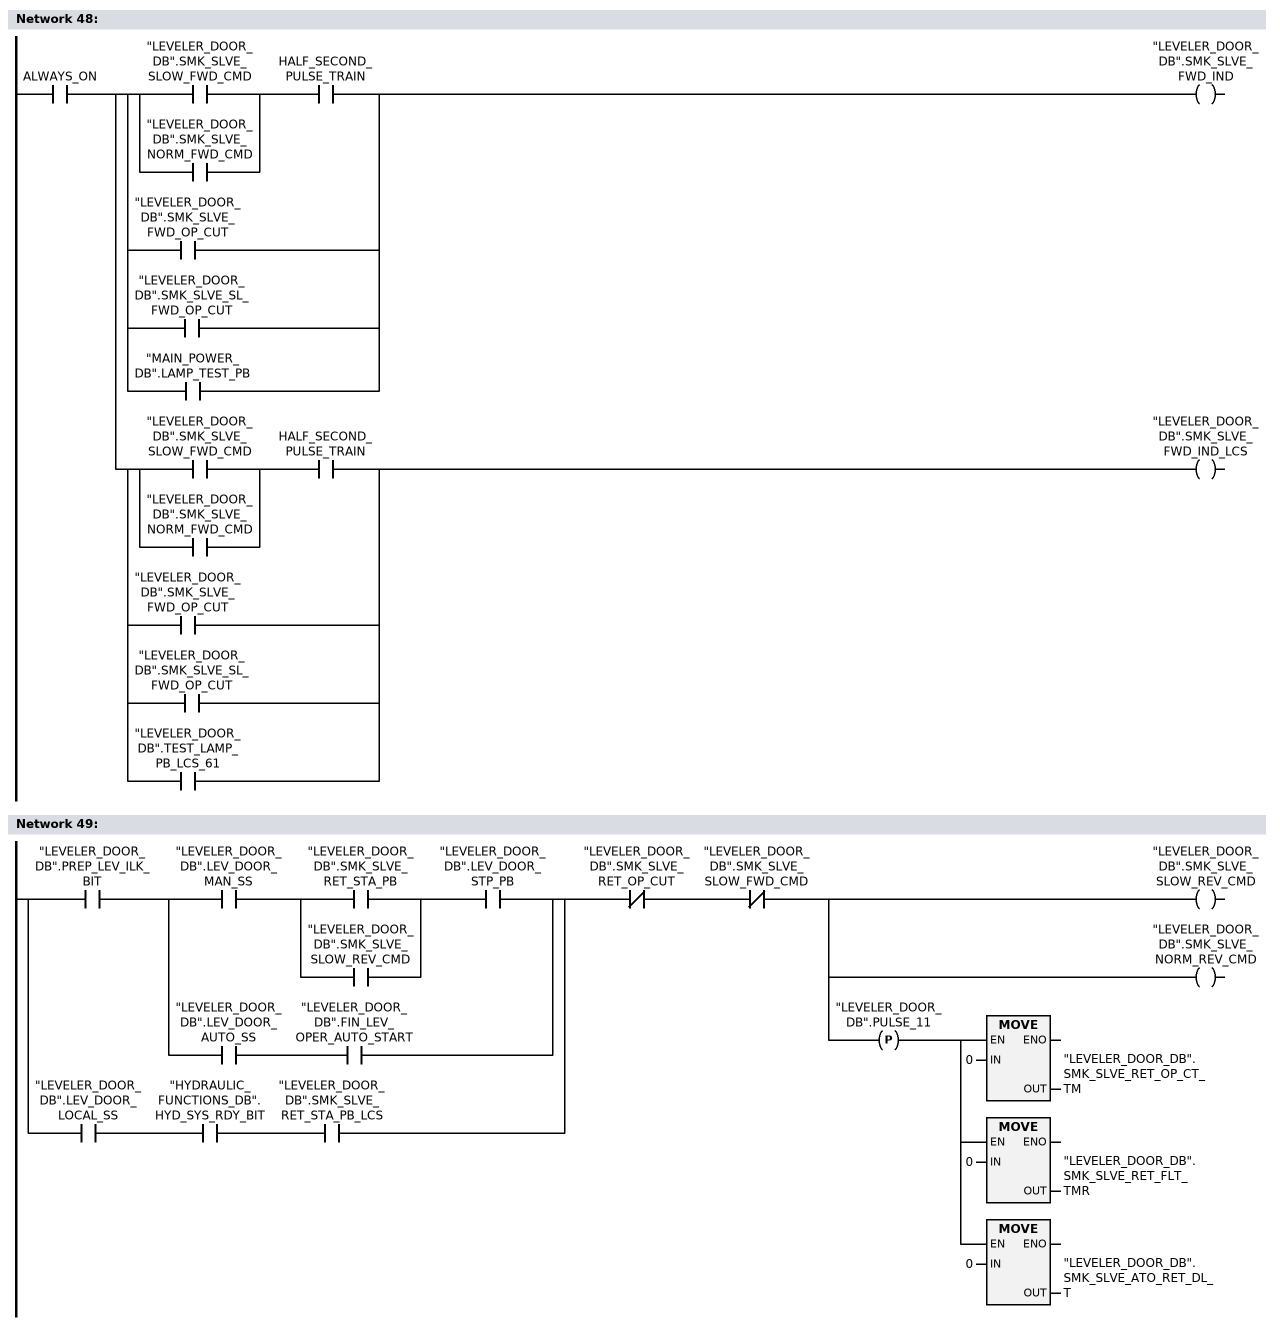
NETWORK
TITLE =
      A     "ALWAYS_ON";
      =     L 0.0;
      A     L 0.0;
      A(;
      A(;
      O     "LEVELER_DOOR_DB".SMK_SLVE_SLOW_FWD_CMD;
      O     "LEVELER_DOOR_DB".SMK_SLVE_NORM_FWD_CMD;
      );
      A     "HALF_SECOND_PULSE_TRAIN";
      O     "LEVELER_DOOR_DB".SMK_SLVE_FWD_OP_CUT;
      O     "LEVELER_DOOR_DB".SMK_SLVE_SL_FWD_OP_CUT;
      O     "MAIN_POWER_DB".LAMP_TEST_PB;
      );
      =     "LEVELER_DOOR_DB".SMK_SLVE_FWD_IND;
      A     L 0.0;
      A(;
      A(;
      O     "LEVELER_DOOR_DB".SMK_SLVE_SLOW_FWD_CMD;
      O     "LEVELER_DOOR_DB".SMK_SLVE_NORM_FWD_CMD;
      );
      A     "HALF_SECOND_PULSE_TRAIN";
      O     "LEVELER_DOOR_DB".SMK_SLVE_FWD_OP_CUT;
      O     "LEVELER_DOOR_DB".SMK_SLVE_SL_FWD_OP_CUT;
      O     "LEVELER_DOOR_DB".TEST_LAMP_PB_LCS_61;
      );
      =     "LEVELER_DOOR_DB".SMK_SLVE_FWD_IND_LCS;
NETWORK
TITLE =
      A(;
      A     "LEVELER_DOOR_DB".PREP_LEV_ILK_BIT;
      A(;
      A     "LEVELER_DOOR_DB".LEV_DOOR_MAN_SS;
      A(;
      O     "LEVELER_DOOR_DB".SMK_SLVE_RET_STA_PB;
      O     "LEVELER_DOOR_DB".SMK_SLVE_SLOW_REV_CMD;
      );
      A     "LEVELER_DOOR_DB".LEV_DOOR_STP_PB;
      O;
      A     "LEVELER_DOOR_DB".LEV_DOOR_AUTO_SS;
      A     "LEVELER_DOOR_DB".FIN_LEV_OPER_AUTO_START;
      );
      O;
      A     "LEVELER_DOOR_DB".LEV_DOOR_LOCAL_SS;
      A     "HYDRAULIC_FUNCTIONS_DB".HYD_SYS_RDY_BIT;
      A     "LEVELER_DOOR_DB".SMK_SLVE_RET_STA_PB_LCS;
      );
      AN    "LEVELER_DOOR_DB".SMK_SLVE_RET_OP_CUT;
      AN    "LEVELER_DOOR_DB".SMK_SLVE_SLOW_FWD_CMD;
      =     L 0.0;
      A     L 0.0;
      BLD   102;
      =     "LEVELER_DOOR_DB".SMK_SLVE_SLOW_REV_CMD;
      A     L 0.0;
      BLD   102;
      =     "LEVELER_DOOR_DB".SMK_SLVE_NORM_REV_CMD;
      A     L 0.0;
      FP    "LEVELER_DOOR_DB".PULSE_11;
      =     L 0.1;
      A     L 0.1;
      JNB   _030;
      L     0;
      T     "LEVELER_DOOR_DB".SMK_SLVE_RET_OP_CT_TM;
_030: NOP   0;
      A     L 0.1;
      JNB   _031;
      L     0;
      T     "LEVELER_DOOR_DB".SMK_SLVE_RET_FLT_TMR;
_031: NOP   0;
      A     L 0.1;
      JNB   _032;
      L     0;
      T     "LEVELER_DOOR_DB".SMK_SLVE_ATO_RET_DL_T;
_032: NOP   0;
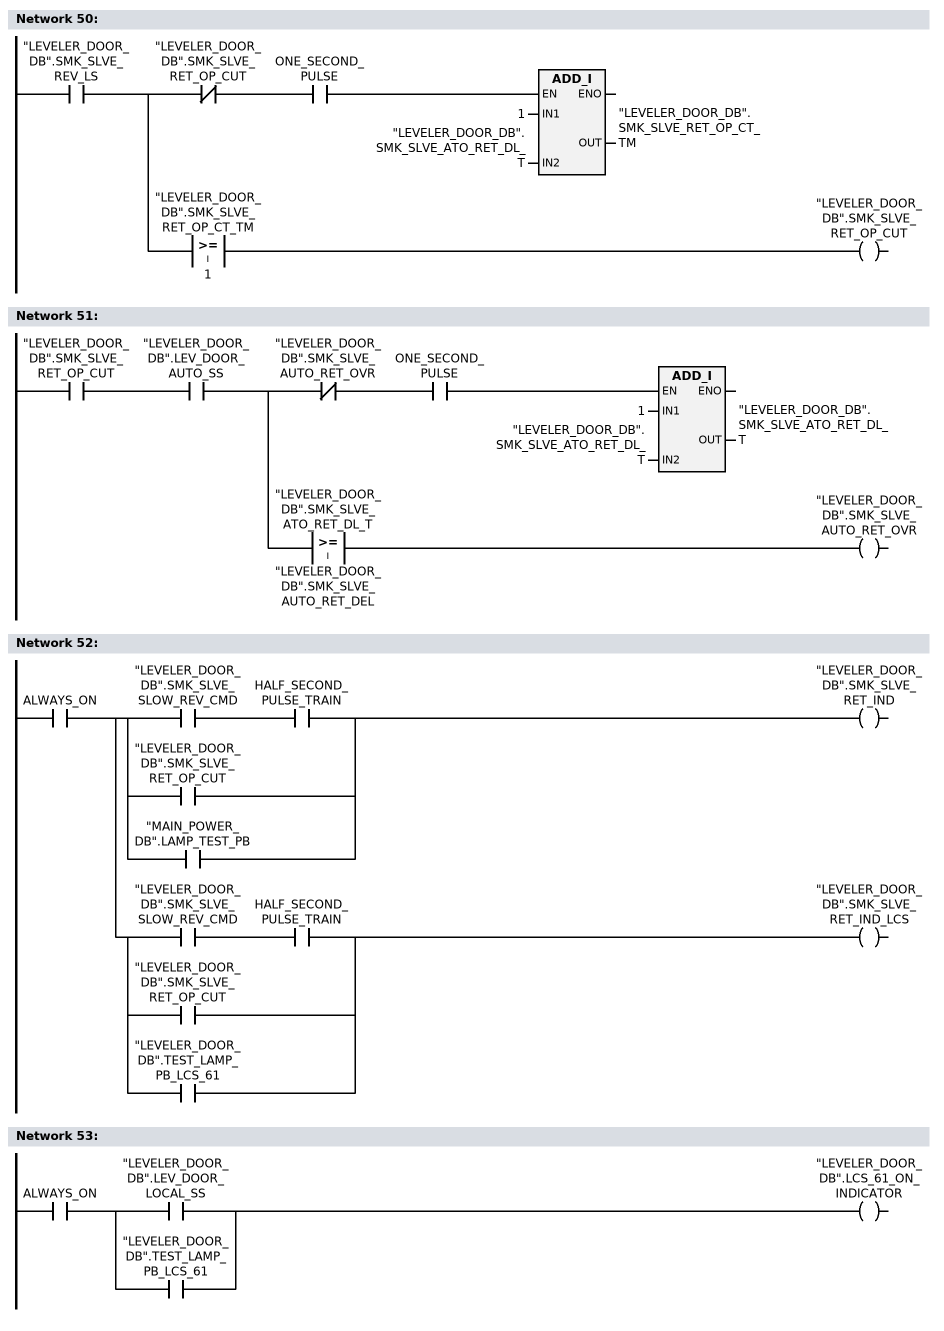
NETWORK
TITLE =
      A     "LEVELER_DOOR_DB".SMK_SLVE_REV_LS;
      =     L 0.0;
      A     L 0.0;
      AN    "LEVELER_DOOR_DB".SMK_SLVE_RET_OP_CUT;
      A     "ONE_SECOND_PULSE";
      JNB   _033;
      L     1;
      L     "LEVELER_DOOR_DB".SMK_SLVE_ATO_RET_DL_T;
      +I;
      T     "LEVELER_DOOR_DB".SMK_SLVE_RET_OP_CT_TM;
_033: NOP   0;
      A     L 0.0;
      A(;
      L     "LEVELER_DOOR_DB".SMK_SLVE_RET_OP_CT_TM;
      L     1;
      >=I;
      );
      =     "LEVELER_DOOR_DB".SMK_SLVE_RET_OP_CUT;
NETWORK
TITLE =
      A     "LEVELER_DOOR_DB".SMK_SLVE_RET_OP_CUT;
      A     "LEVELER_DOOR_DB".LEV_DOOR_AUTO_SS;
      =     L 0.0;
      A     L 0.0;
      AN    "LEVELER_DOOR_DB".SMK_SLVE_AUTO_RET_OVR;
      A     "ONE_SECOND_PULSE";
      JNB   _034;
      L     1;
      L     "LEVELER_DOOR_DB".SMK_SLVE_ATO_RET_DL_T;
      +I;
      T     "LEVELER_DOOR_DB".SMK_SLVE_ATO_RET_DL_T;
_034: NOP   0;
      A     L 0.0;
      A(;
      L     "LEVELER_DOOR_DB".SMK_SLVE_ATO_RET_DL_T;
      L     "LEVELER_DOOR_DB".SMK_SLVE_AUTO_RET_DEL;
      >=I;
      );
      =     "LEVELER_DOOR_DB".SMK_SLVE_AUTO_RET_OVR;
NETWORK
TITLE =
      A     "ALWAYS_ON";
      =     L 0.0;
      A     L 0.0;
      A(;
      A     "LEVELER_DOOR_DB".SMK_SLVE_SLOW_REV_CMD;
      A     "HALF_SECOND_PULSE_TRAIN";
      O     "LEVELER_DOOR_DB".SMK_SLVE_RET_OP_CUT;
      O     "MAIN_POWER_DB".LAMP_TEST_PB;
      );
      =     "LEVELER_DOOR_DB".SMK_SLVE_RET_IND;
      A     L 0.0;
      A(;
      A     "LEVELER_DOOR_DB".SMK_SLVE_SLOW_REV_CMD;
      A     "HALF_SECOND_PULSE_TRAIN";
      O     "LEVELER_DOOR_DB".SMK_SLVE_RET_OP_CUT;
      O     "LEVELER_DOOR_DB".TEST_LAMP_PB_LCS_61;
      );
      =     "LEVELER_DOOR_DB".SMK_SLVE_RET_IND_LCS;
NETWORK
TITLE =
      A     "ALWAYS_ON";
      A(;
      O     "LEVELER_DOOR_DB".LEV_DOOR_LOCAL_SS;
      O     "LEVELER_DOOR_DB".TEST_LAMP_PB_LCS_61;
      );
      =     "LEVELER_DOOR_DB".LCS_61_ON_INDICATOR;
END_FUNCTION

FUNCTION "TRAVEL_DRIVE" : VOID	// FC 7
AUTHOR : Kamillas
VERSION : 0.1
BEGIN
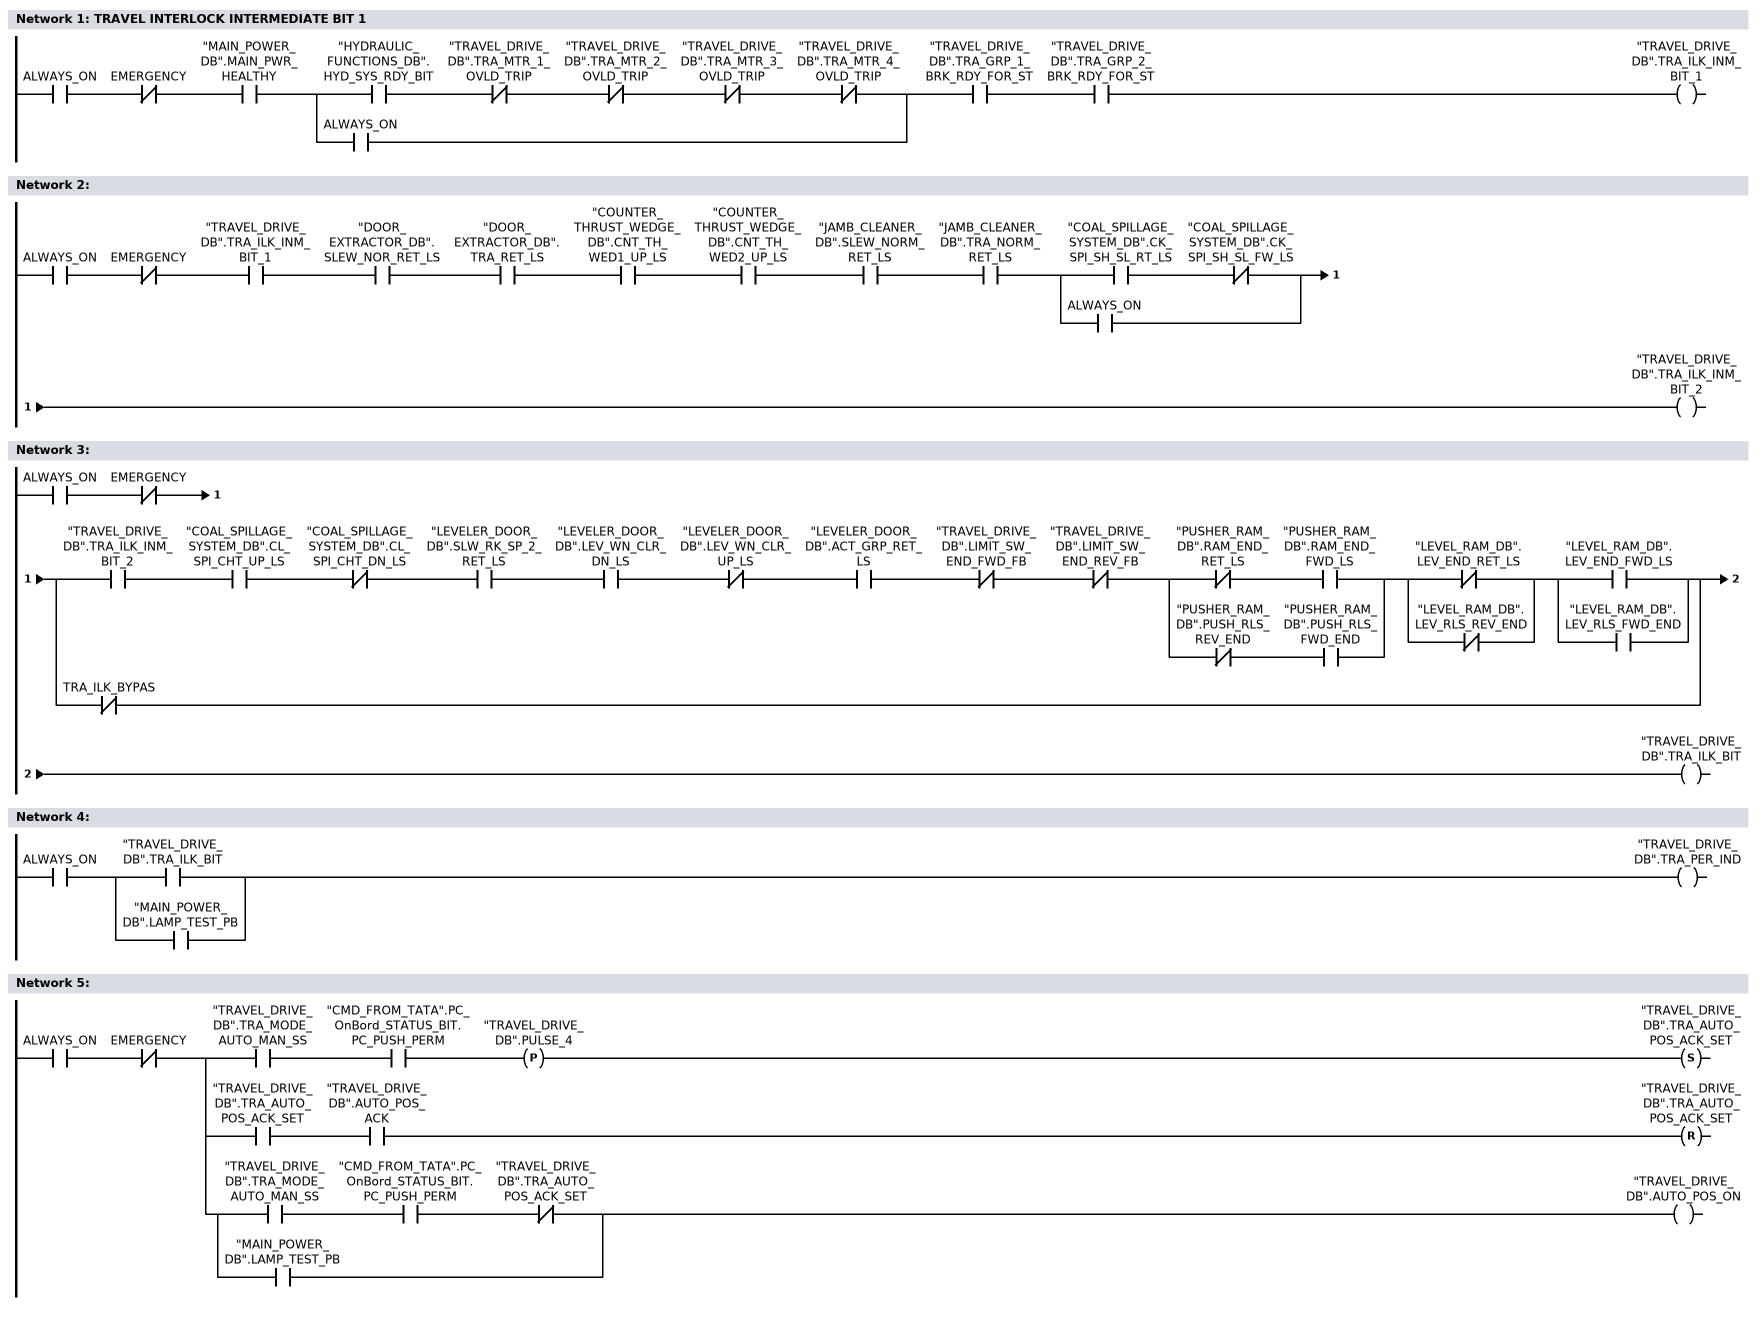
NETWORK
TITLE = TRAVEL INTERLOCK INTERMEDIATE BIT 1
      A     "ALWAYS_ON";
      AN    "EMERGENCY";
      A     "MAIN_POWER_DB".MAIN_PWR_HEALTHY;
      A(;
      A     "HYDRAULIC_FUNCTIONS_DB".HYD_SYS_RDY_BIT;
      AN    "TRAVEL_DRIVE_DB".TRA_MTR_1_OVLD_TRIP;
      AN    "TRAVEL_DRIVE_DB".TRA_MTR_2_OVLD_TRIP;
      AN    "TRAVEL_DRIVE_DB".TRA_MTR_3_OVLD_TRIP;
      AN    "TRAVEL_DRIVE_DB".TRA_MTR_4_OVLD_TRIP;
      O     "ALWAYS_ON";
      );
      A     "TRAVEL_DRIVE_DB".TRA_GRP_1_BRK_RDY_FOR_ST;
      A     "TRAVEL_DRIVE_DB".TRA_GRP_2_BRK_RDY_FOR_ST;
      =     "TRAVEL_DRIVE_DB".TRA_ILK_INM_BIT_1;
NETWORK
TITLE =
      A     "ALWAYS_ON";
      AN    "EMERGENCY";
      A     "TRAVEL_DRIVE_DB".TRA_ILK_INM_BIT_1;
      A     "DOOR_EXTRACTOR_DB".SLEW_NOR_RET_LS;
      A     "DOOR_EXTRACTOR_DB".TRA_RET_LS;
      A     "COUNTER_THRUST_WEDGE_DB".CNT_TH_WED1_UP_LS;
      A     "COUNTER_THRUST_WEDGE_DB".CNT_TH_WED2_UP_LS;
      A     "JAMB_CLEANER_DB".SLEW_NORM_RET_LS;
      A     "JAMB_CLEANER_DB".TRA_NORM_RET_LS;
      A(;
      A     "COAL_SPILLAGE_SYSTEM_DB".CK_SPI_SH_SL_RT_LS;
      AN    "COAL_SPILLAGE_SYSTEM_DB".CK_SPI_SH_SL_FW_LS;
      O     "ALWAYS_ON";
      );
      =     "TRAVEL_DRIVE_DB".TRA_ILK_INM_BIT_2;
NETWORK
TITLE =
      A     "ALWAYS_ON";
      AN    "EMERGENCY";
      A(;
      A     "TRAVEL_DRIVE_DB".TRA_ILK_INM_BIT_2;
      A     "COAL_SPILLAGE_SYSTEM_DB".CL_SPI_CHT_UP_LS;
      AN    "COAL_SPILLAGE_SYSTEM_DB".CL_SPI_CHT_DN_LS;
      A     "LEVELER_DOOR_DB".SLW_RK_SP_2_RET_LS;
      A     "LEVELER_DOOR_DB".LEV_WN_CLR_DN_LS;
      AN    "LEVELER_DOOR_DB".LEV_WN_CLR_UP_LS;
      A     "LEVELER_DOOR_DB".ACT_GRP_RET_LS;
      AN    "TRAVEL_DRIVE_DB".LIMIT_SW_END_FWD_FB;
      AN    "TRAVEL_DRIVE_DB".LIMIT_SW_END_REV_FB;
      A(;
      AN    "PUSHER_RAM_DB".RAM_END_RET_LS;
      A     "PUSHER_RAM_DB".RAM_END_FWD_LS;
      O;
      AN    "PUSHER_RAM_DB".PUSH_RLS_REV_END;
      A     "PUSHER_RAM_DB".PUSH_RLS_FWD_END;
      );
      A(;
      ON    "LEVEL_RAM_DB".LEV_END_RET_LS;
      ON    "LEVEL_RAM_DB".LEV_RLS_REV_END;
      );
      A(;
      O     "LEVEL_RAM_DB".LEV_END_FWD_LS;
      O     "LEVEL_RAM_DB".LEV_RLS_FWD_END;
      );
      ON    "TRA_ILK_BYPAS";
      );
      =     "TRAVEL_DRIVE_DB".TRA_ILK_BIT;
NETWORK
TITLE =
      A     "ALWAYS_ON";
      A(;
      O     "TRAVEL_DRIVE_DB".TRA_ILK_BIT;
      O     "MAIN_POWER_DB".LAMP_TEST_PB;
      );
      =     "TRAVEL_DRIVE_DB".TRA_PER_IND;
NETWORK
TITLE =
      A     "ALWAYS_ON";
      AN    "EMERGENCY";
      =     L 0.0;
      A     L 0.0;
      A     "TRAVEL_DRIVE_DB".TRA_MODE_AUTO_MAN_SS;
      A     "CMD_FROM_TATA".PC_OnBord_STATUS_BIT.PC_PUSH_PERM;
      FP    "TRAVEL_DRIVE_DB".PULSE_4;
      S     "TRAVEL_DRIVE_DB".TRA_AUTO_POS_ACK_SET;
      A     L 0.0;
      A     "TRAVEL_DRIVE_DB".TRA_AUTO_POS_ACK_SET;
      A     "TRAVEL_DRIVE_DB".AUTO_POS_ACK;
      R     "TRAVEL_DRIVE_DB".TRA_AUTO_POS_ACK_SET;
      A     L 0.0;
      A(;
      A     "TRAVEL_DRIVE_DB".TRA_MODE_AUTO_MAN_SS;
      A     "CMD_FROM_TATA".PC_OnBord_STATUS_BIT.PC_PUSH_PERM;
      AN    "TRAVEL_DRIVE_DB".TRA_AUTO_POS_ACK_SET;
      O     "MAIN_POWER_DB".LAMP_TEST_PB;
      );
      =     "TRAVEL_DRIVE_DB".AUTO_POS_ON;
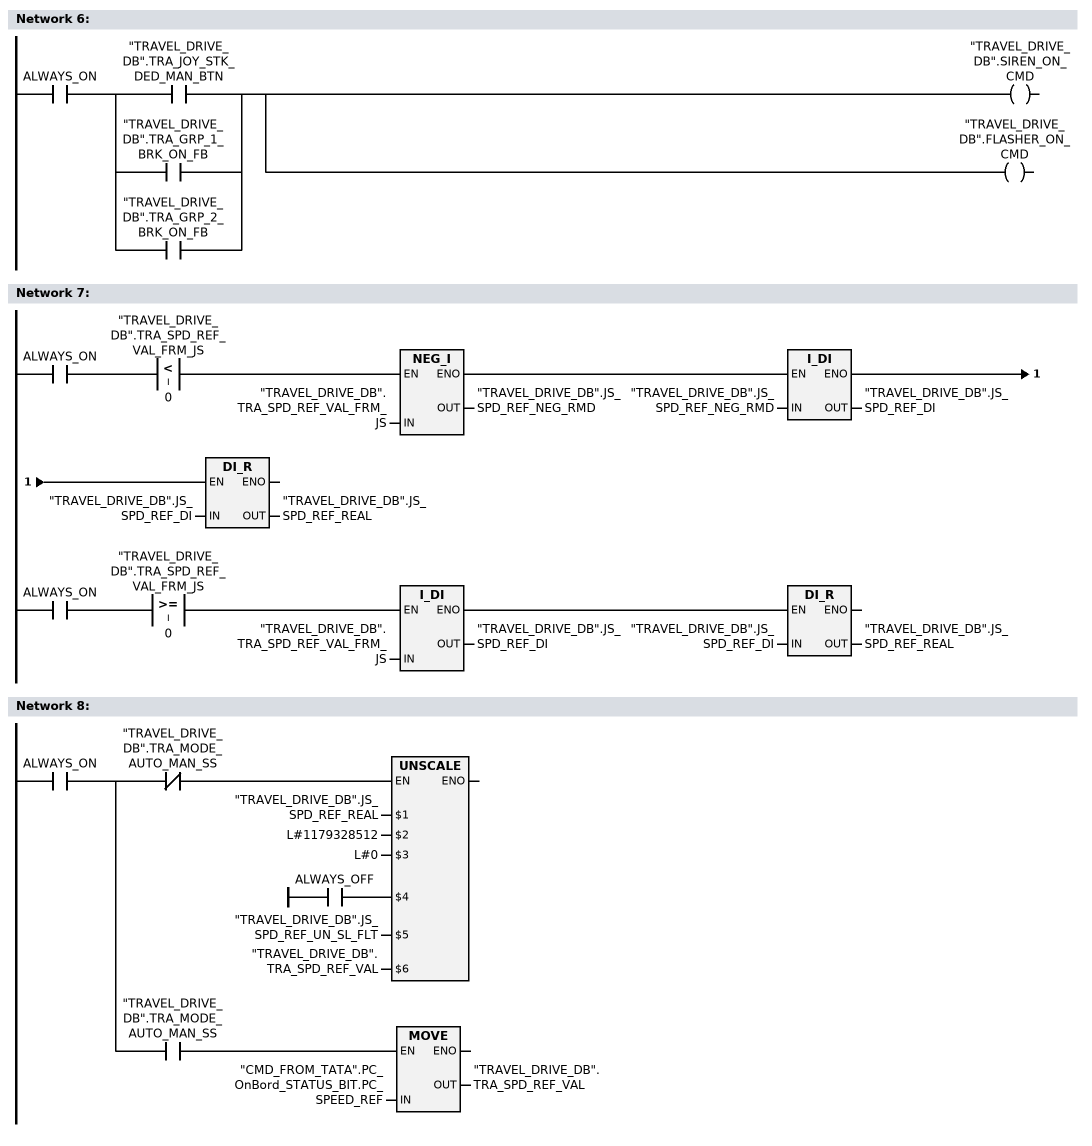
NETWORK
TITLE =
      A     "ALWAYS_ON";
      A(;
      O     "TRAVEL_DRIVE_DB".TRA_JOY_STK_DED_MAN_BTN;
      O     "TRAVEL_DRIVE_DB".TRA_GRP_1_BRK_ON_FB;
      O     "TRAVEL_DRIVE_DB".TRA_GRP_2_BRK_ON_FB;
      );
      =     "TRAVEL_DRIVE_DB".SIREN_ON_CMD;
      =     "TRAVEL_DRIVE_DB".FLASHER_ON_CMD;
NETWORK
TITLE =
      A     "ALWAYS_ON";
      =     L 0.0;
      A(;
      A(;
      A     L 0.0;
      A(;
      L     "TRAVEL_DRIVE_DB".TRA_SPD_REF_VAL_FRM_JS;
      L     0;
      <I;
      );
      JNB   _001;
      L     "TRAVEL_DRIVE_DB".TRA_SPD_REF_VAL_FRM_JS;
      NEGI;
      T     "TRAVEL_DRIVE_DB".JS_SPD_REF_NEG_RMD;
      AN    OV;
      SAVE;
      CLR;
_001: A     BR;
      );
      JNB   _002;
      L     "TRAVEL_DRIVE_DB".JS_SPD_REF_NEG_RMD;
      ITD;
      T     "TRAVEL_DRIVE_DB".JS_SPD_REF_DI;
      SET;
      SAVE;
      CLR;
_002: A     BR;
      );
      JNB   _003;
      L     "TRAVEL_DRIVE_DB".JS_SPD_REF_DI;
      DTR;
      T     "TRAVEL_DRIVE_DB".JS_SPD_REF_REAL;
_003: NOP   0;
      A(;
      A     L 0.0;
      A(;
      L     "TRAVEL_DRIVE_DB".TRA_SPD_REF_VAL_FRM_JS;
      L     0;
      >=I;
      );
      JNB   _004;
      L     "TRAVEL_DRIVE_DB".TRA_SPD_REF_VAL_FRM_JS;
      ITD;
      T     "TRAVEL_DRIVE_DB".JS_SPD_REF_DI;
      SET;
      SAVE;
      CLR;
_004: A     BR;
      );
      JNB   _005;
      L     "TRAVEL_DRIVE_DB".JS_SPD_REF_DI;
      DTR;
      T     "TRAVEL_DRIVE_DB".JS_SPD_REF_REAL;
_005: NOP   0;
NETWORK
TITLE =
      A     "ALWAYS_ON";
      =     L 0.0;
      A     "ALWAYS_OFF";
      =     L 0.1;
      BLD   103;
      A     L 0.0;
      AN    "TRAVEL_DRIVE_DB".TRA_MODE_AUTO_MAN_SS;
      JNB   _006;
      CALL  "UNSCALE" (
           $1                       := "TRAVEL_DRIVE_DB".JS_SPD_REF_REAL,
           $2                       := L#1179328512,
           $3                       := L#0,
           $4                       := L 0.1,
           $5                       := "TRAVEL_DRIVE_DB".JS_SPD_REF_UN_SL_FLT,
           $6                       := "TRAVEL_DRIVE_DB".TRA_SPD_REF_VAL);
_006: NOP   0;
      A     L 0.0;
      A     "TRAVEL_DRIVE_DB".TRA_MODE_AUTO_MAN_SS;
      JNB   _007;
      L     "CMD_FROM_TATA".PC_OnBord_STATUS_BIT.PC_SPEED_REF;
      T     "TRAVEL_DRIVE_DB".TRA_SPD_REF_VAL;
_007: NOP   0;
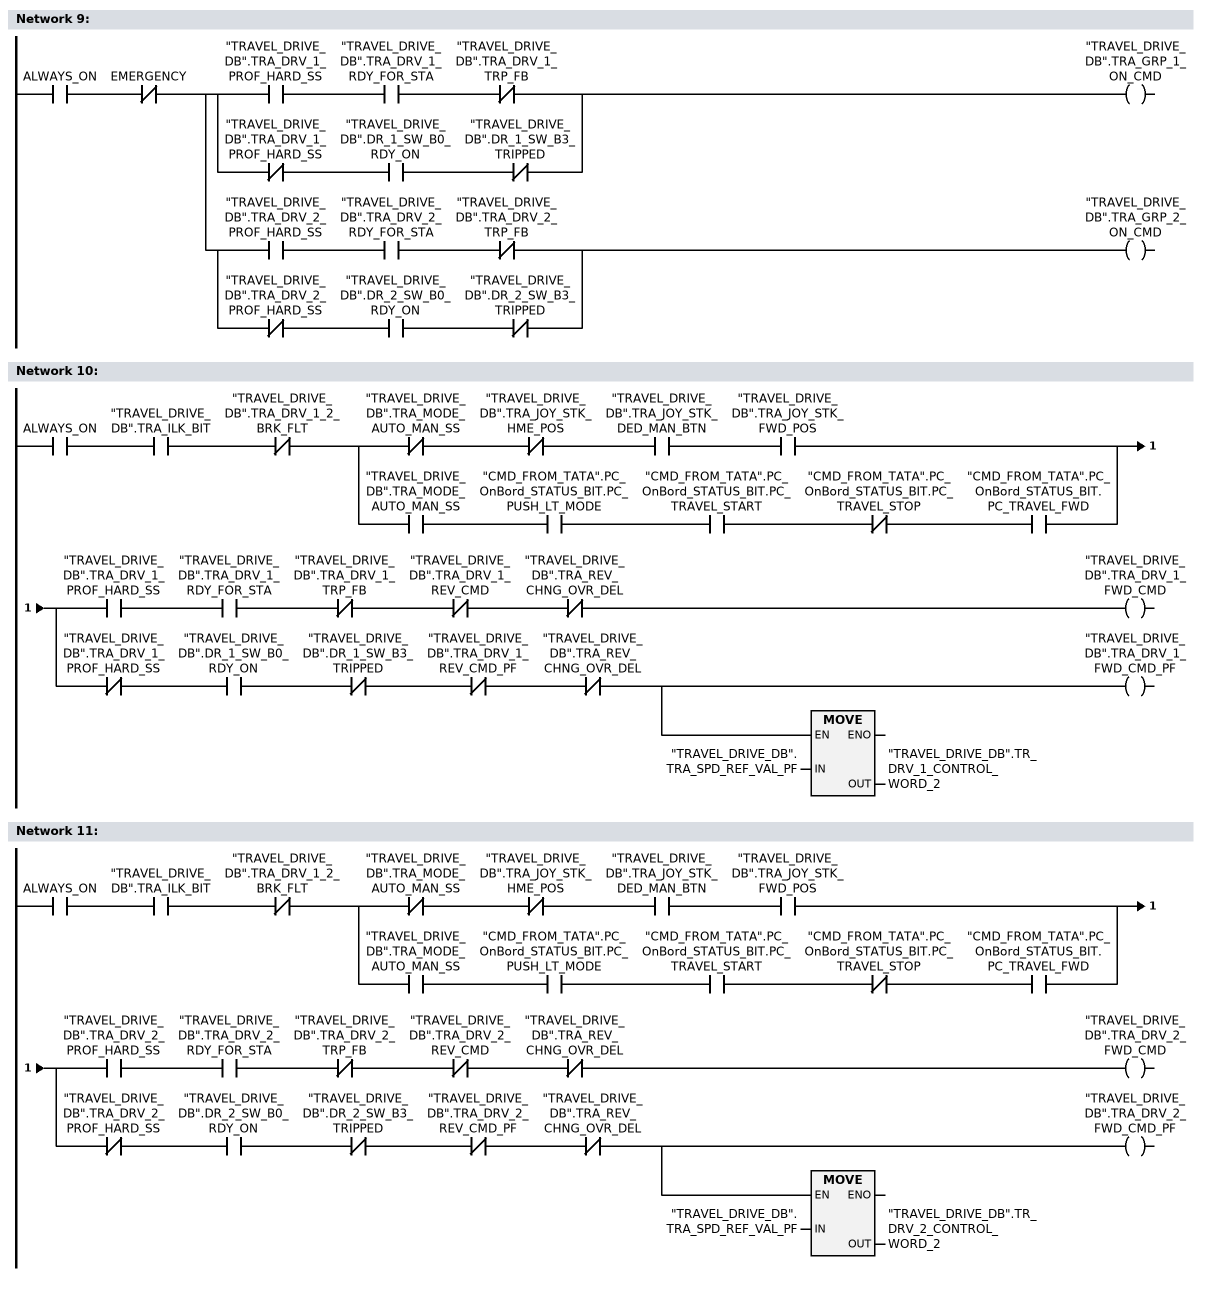
NETWORK
TITLE =
      A     "ALWAYS_ON";
      AN    "EMERGENCY";
      =     L 0.0;
      A     L 0.0;
      A(;
      A     "TRAVEL_DRIVE_DB".TRA_DRV_1_PROF_HARD_SS;
      A     "TRAVEL_DRIVE_DB".TRA_DRV_1_RDY_FOR_STA;
      AN    "TRAVEL_DRIVE_DB".TRA_DRV_1_TRP_FB;
      O;
      AN    "TRAVEL_DRIVE_DB".TRA_DRV_1_PROF_HARD_SS;
      A     "TRAVEL_DRIVE_DB".DR_1_SW_B0_RDY_ON;
      AN    "TRAVEL_DRIVE_DB".DR_1_SW_B3_TRIPPED;
      );
      =     "TRAVEL_DRIVE_DB".TRA_GRP_1_ON_CMD;
      A     L 0.0;
      A(;
      A     "TRAVEL_DRIVE_DB".TRA_DRV_2_PROF_HARD_SS;
      A     "TRAVEL_DRIVE_DB".TRA_DRV_2_RDY_FOR_STA;
      AN    "TRAVEL_DRIVE_DB".TRA_DRV_2_TRP_FB;
      O;
      AN    "TRAVEL_DRIVE_DB".TRA_DRV_2_PROF_HARD_SS;
      A     "TRAVEL_DRIVE_DB".DR_2_SW_B0_RDY_ON;
      AN    "TRAVEL_DRIVE_DB".DR_2_SW_B3_TRIPPED;
      );
      =     "TRAVEL_DRIVE_DB".TRA_GRP_2_ON_CMD;
NETWORK
TITLE =
      A     "ALWAYS_ON";
      A     "TRAVEL_DRIVE_DB".TRA_ILK_BIT;
      AN    "TRAVEL_DRIVE_DB".TRA_DRV_1_2_BRK_FLT;
      A(;
      AN    "TRAVEL_DRIVE_DB".TRA_MODE_AUTO_MAN_SS;
      AN    "TRAVEL_DRIVE_DB".TRA_JOY_STK_HME_POS;
      A     "TRAVEL_DRIVE_DB".TRA_JOY_STK_DED_MAN_BTN;
      A     "TRAVEL_DRIVE_DB".TRA_JOY_STK_FWD_POS;
      O;
      A     "TRAVEL_DRIVE_DB".TRA_MODE_AUTO_MAN_SS;
      A     "CMD_FROM_TATA".PC_OnBord_STATUS_BIT.PC_PUSH_LT_MODE;
      A     "CMD_FROM_TATA".PC_OnBord_STATUS_BIT.PC_TRAVEL_START;
      AN    "CMD_FROM_TATA".PC_OnBord_STATUS_BIT.PC_TRAVEL_STOP;
      A     "CMD_FROM_TATA".PC_OnBord_STATUS_BIT.PC_TRAVEL_FWD;
      );
      =     L 0.0;
      A     L 0.0;
      A     "TRAVEL_DRIVE_DB".TRA_DRV_1_PROF_HARD_SS;
      A     "TRAVEL_DRIVE_DB".TRA_DRV_1_RDY_FOR_STA;
      AN    "TRAVEL_DRIVE_DB".TRA_DRV_1_TRP_FB;
      AN    "TRAVEL_DRIVE_DB".TRA_DRV_1_REV_CMD;
      AN    "TRAVEL_DRIVE_DB".TRA_REV_CHNG_OVR_DEL;
      =     "TRAVEL_DRIVE_DB".TRA_DRV_1_FWD_CMD;
      A     L 0.0;
      AN    "TRAVEL_DRIVE_DB".TRA_DRV_1_PROF_HARD_SS;
      A     "TRAVEL_DRIVE_DB".DR_1_SW_B0_RDY_ON;
      AN    "TRAVEL_DRIVE_DB".DR_1_SW_B3_TRIPPED;
      AN    "TRAVEL_DRIVE_DB".TRA_DRV_1_REV_CMD_PF;
      AN    "TRAVEL_DRIVE_DB".TRA_REV_CHNG_OVR_DEL;
      =     L 0.1;
      A     L 0.1;
      BLD   102;
      =     "TRAVEL_DRIVE_DB".TRA_DRV_1_FWD_CMD_PF;
      A     L 0.1;
      JNB   _008;
      L     "TRAVEL_DRIVE_DB".TRA_SPD_REF_VAL_PF;
      T     "TRAVEL_DRIVE_DB".TR_DRV_1_CONTROL_WORD_2;
_008: NOP   0;
NETWORK
TITLE =
      A     "ALWAYS_ON";
      A     "TRAVEL_DRIVE_DB".TRA_ILK_BIT;
      AN    "TRAVEL_DRIVE_DB".TRA_DRV_1_2_BRK_FLT;
      A(;
      AN    "TRAVEL_DRIVE_DB".TRA_MODE_AUTO_MAN_SS;
      AN    "TRAVEL_DRIVE_DB".TRA_JOY_STK_HME_POS;
      A     "TRAVEL_DRIVE_DB".TRA_JOY_STK_DED_MAN_BTN;
      A     "TRAVEL_DRIVE_DB".TRA_JOY_STK_FWD_POS;
      O;
      A     "TRAVEL_DRIVE_DB".TRA_MODE_AUTO_MAN_SS;
      A     "CMD_FROM_TATA".PC_OnBord_STATUS_BIT.PC_PUSH_LT_MODE;
      A     "CMD_FROM_TATA".PC_OnBord_STATUS_BIT.PC_TRAVEL_START;
      AN    "CMD_FROM_TATA".PC_OnBord_STATUS_BIT.PC_TRAVEL_STOP;
      A     "CMD_FROM_TATA".PC_OnBord_STATUS_BIT.PC_TRAVEL_FWD;
      );
      =     L 0.0;
      A     L 0.0;
      A     "TRAVEL_DRIVE_DB".TRA_DRV_2_PROF_HARD_SS;
      A     "TRAVEL_DRIVE_DB".TRA_DRV_2_RDY_FOR_STA;
      AN    "TRAVEL_DRIVE_DB".TRA_DRV_2_TRP_FB;
      AN    "TRAVEL_DRIVE_DB".TRA_DRV_2_REV_CMD;
      AN    "TRAVEL_DRIVE_DB".TRA_REV_CHNG_OVR_DEL;
      =     "TRAVEL_DRIVE_DB".TRA_DRV_2_FWD_CMD;
      A     L 0.0;
      AN    "TRAVEL_DRIVE_DB".TRA_DRV_2_PROF_HARD_SS;
      A     "TRAVEL_DRIVE_DB".DR_2_SW_B0_RDY_ON;
      AN    "TRAVEL_DRIVE_DB".DR_2_SW_B3_TRIPPED;
      AN    "TRAVEL_DRIVE_DB".TRA_DRV_2_REV_CMD_PF;
      AN    "TRAVEL_DRIVE_DB".TRA_REV_CHNG_OVR_DEL;
      =     L 0.1;
      A     L 0.1;
      BLD   102;
      =     "TRAVEL_DRIVE_DB".TRA_DRV_2_FWD_CMD_PF;
      A     L 0.1;
      JNB   _009;
      L     "TRAVEL_DRIVE_DB".TRA_SPD_REF_VAL_PF;
      T     "TRAVEL_DRIVE_DB".TR_DRV_2_CONTROL_WORD_2;
_009: NOP   0;
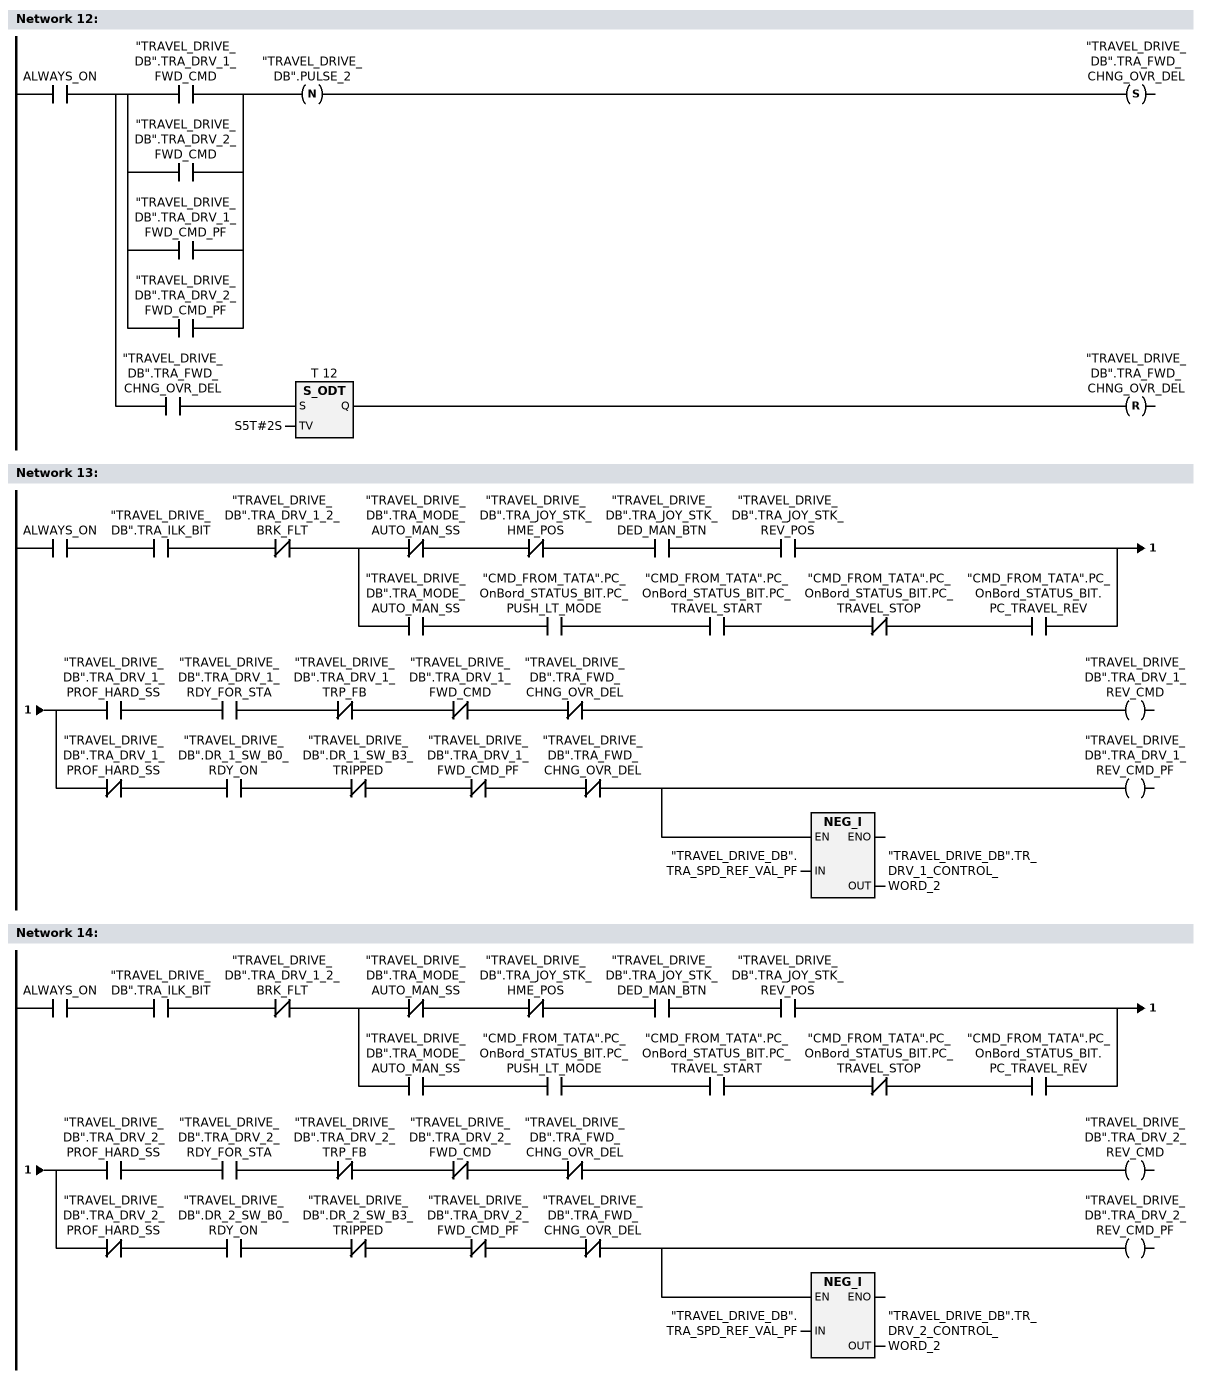
NETWORK
TITLE =
      A     "ALWAYS_ON";
      =     L 0.0;
      A     L 0.0;
      A(;
      O     "TRAVEL_DRIVE_DB".TRA_DRV_1_FWD_CMD;
      O     "TRAVEL_DRIVE_DB".TRA_DRV_2_FWD_CMD;
      O     "TRAVEL_DRIVE_DB".TRA_DRV_1_FWD_CMD_PF;
      O     "TRAVEL_DRIVE_DB".TRA_DRV_2_FWD_CMD_PF;
      );
      FN    "TRAVEL_DRIVE_DB".PULSE_2;
      S     "TRAVEL_DRIVE_DB".TRA_FWD_CHNG_OVR_DEL;
      A     L 0.0;
      A     "TRAVEL_DRIVE_DB".TRA_FWD_CHNG_OVR_DEL;
      L     S5T#2S;
      SD    T 12;
      NOP   0;
      NOP   0;
      NOP   0;
      A     T 12;
      R     "TRAVEL_DRIVE_DB".TRA_FWD_CHNG_OVR_DEL;
NETWORK
TITLE =
      A     "ALWAYS_ON";
      A     "TRAVEL_DRIVE_DB".TRA_ILK_BIT;
      AN    "TRAVEL_DRIVE_DB".TRA_DRV_1_2_BRK_FLT;
      A(;
      AN    "TRAVEL_DRIVE_DB".TRA_MODE_AUTO_MAN_SS;
      AN    "TRAVEL_DRIVE_DB".TRA_JOY_STK_HME_POS;
      A     "TRAVEL_DRIVE_DB".TRA_JOY_STK_DED_MAN_BTN;
      A     "TRAVEL_DRIVE_DB".TRA_JOY_STK_REV_POS;
      O;
      A     "TRAVEL_DRIVE_DB".TRA_MODE_AUTO_MAN_SS;
      A     "CMD_FROM_TATA".PC_OnBord_STATUS_BIT.PC_PUSH_LT_MODE;
      A     "CMD_FROM_TATA".PC_OnBord_STATUS_BIT.PC_TRAVEL_START;
      AN    "CMD_FROM_TATA".PC_OnBord_STATUS_BIT.PC_TRAVEL_STOP;
      A     "CMD_FROM_TATA".PC_OnBord_STATUS_BIT.PC_TRAVEL_REV;
      );
      =     L 0.0;
      A     L 0.0;
      A     "TRAVEL_DRIVE_DB".TRA_DRV_1_PROF_HARD_SS;
      A     "TRAVEL_DRIVE_DB".TRA_DRV_1_RDY_FOR_STA;
      AN    "TRAVEL_DRIVE_DB".TRA_DRV_1_TRP_FB;
      AN    "TRAVEL_DRIVE_DB".TRA_DRV_1_FWD_CMD;
      AN    "TRAVEL_DRIVE_DB".TRA_FWD_CHNG_OVR_DEL;
      =     "TRAVEL_DRIVE_DB".TRA_DRV_1_REV_CMD;
      A     L 0.0;
      AN    "TRAVEL_DRIVE_DB".TRA_DRV_1_PROF_HARD_SS;
      A     "TRAVEL_DRIVE_DB".DR_1_SW_B0_RDY_ON;
      AN    "TRAVEL_DRIVE_DB".DR_1_SW_B3_TRIPPED;
      AN    "TRAVEL_DRIVE_DB".TRA_DRV_1_FWD_CMD_PF;
      AN    "TRAVEL_DRIVE_DB".TRA_FWD_CHNG_OVR_DEL;
      =     L 0.1;
      A     L 0.1;
      BLD   102;
      =     "TRAVEL_DRIVE_DB".TRA_DRV_1_REV_CMD_PF;
      A     L 0.1;
      JNB   _00a;
      L     "TRAVEL_DRIVE_DB".TRA_SPD_REF_VAL_PF;
      NEGI;
      T     "TRAVEL_DRIVE_DB".TR_DRV_1_CONTROL_WORD_2;
_00a: NOP   0;
NETWORK
TITLE =
      A     "ALWAYS_ON";
      A     "TRAVEL_DRIVE_DB".TRA_ILK_BIT;
      AN    "TRAVEL_DRIVE_DB".TRA_DRV_1_2_BRK_FLT;
      A(;
      AN    "TRAVEL_DRIVE_DB".TRA_MODE_AUTO_MAN_SS;
      AN    "TRAVEL_DRIVE_DB".TRA_JOY_STK_HME_POS;
      A     "TRAVEL_DRIVE_DB".TRA_JOY_STK_DED_MAN_BTN;
      A     "TRAVEL_DRIVE_DB".TRA_JOY_STK_REV_POS;
      O;
      A     "TRAVEL_DRIVE_DB".TRA_MODE_AUTO_MAN_SS;
      A     "CMD_FROM_TATA".PC_OnBord_STATUS_BIT.PC_PUSH_LT_MODE;
      A     "CMD_FROM_TATA".PC_OnBord_STATUS_BIT.PC_TRAVEL_START;
      AN    "CMD_FROM_TATA".PC_OnBord_STATUS_BIT.PC_TRAVEL_STOP;
      A     "CMD_FROM_TATA".PC_OnBord_STATUS_BIT.PC_TRAVEL_REV;
      );
      =     L 0.0;
      A     L 0.0;
      A     "TRAVEL_DRIVE_DB".TRA_DRV_2_PROF_HARD_SS;
      A     "TRAVEL_DRIVE_DB".TRA_DRV_2_RDY_FOR_STA;
      AN    "TRAVEL_DRIVE_DB".TRA_DRV_2_TRP_FB;
      AN    "TRAVEL_DRIVE_DB".TRA_DRV_2_FWD_CMD;
      AN    "TRAVEL_DRIVE_DB".TRA_FWD_CHNG_OVR_DEL;
      =     "TRAVEL_DRIVE_DB".TRA_DRV_2_REV_CMD;
      A     L 0.0;
      AN    "TRAVEL_DRIVE_DB".TRA_DRV_2_PROF_HARD_SS;
      A     "TRAVEL_DRIVE_DB".DR_2_SW_B0_RDY_ON;
      AN    "TRAVEL_DRIVE_DB".DR_2_SW_B3_TRIPPED;
      AN    "TRAVEL_DRIVE_DB".TRA_DRV_2_FWD_CMD_PF;
      AN    "TRAVEL_DRIVE_DB".TRA_FWD_CHNG_OVR_DEL;
      =     L 0.1;
      A     L 0.1;
      BLD   102;
      =     "TRAVEL_DRIVE_DB".TRA_DRV_2_REV_CMD_PF;
      A     L 0.1;
      JNB   _00b;
      L     "TRAVEL_DRIVE_DB".TRA_SPD_REF_VAL_PF;
      NEGI;
      T     "TRAVEL_DRIVE_DB".TR_DRV_2_CONTROL_WORD_2;
_00b: NOP   0;
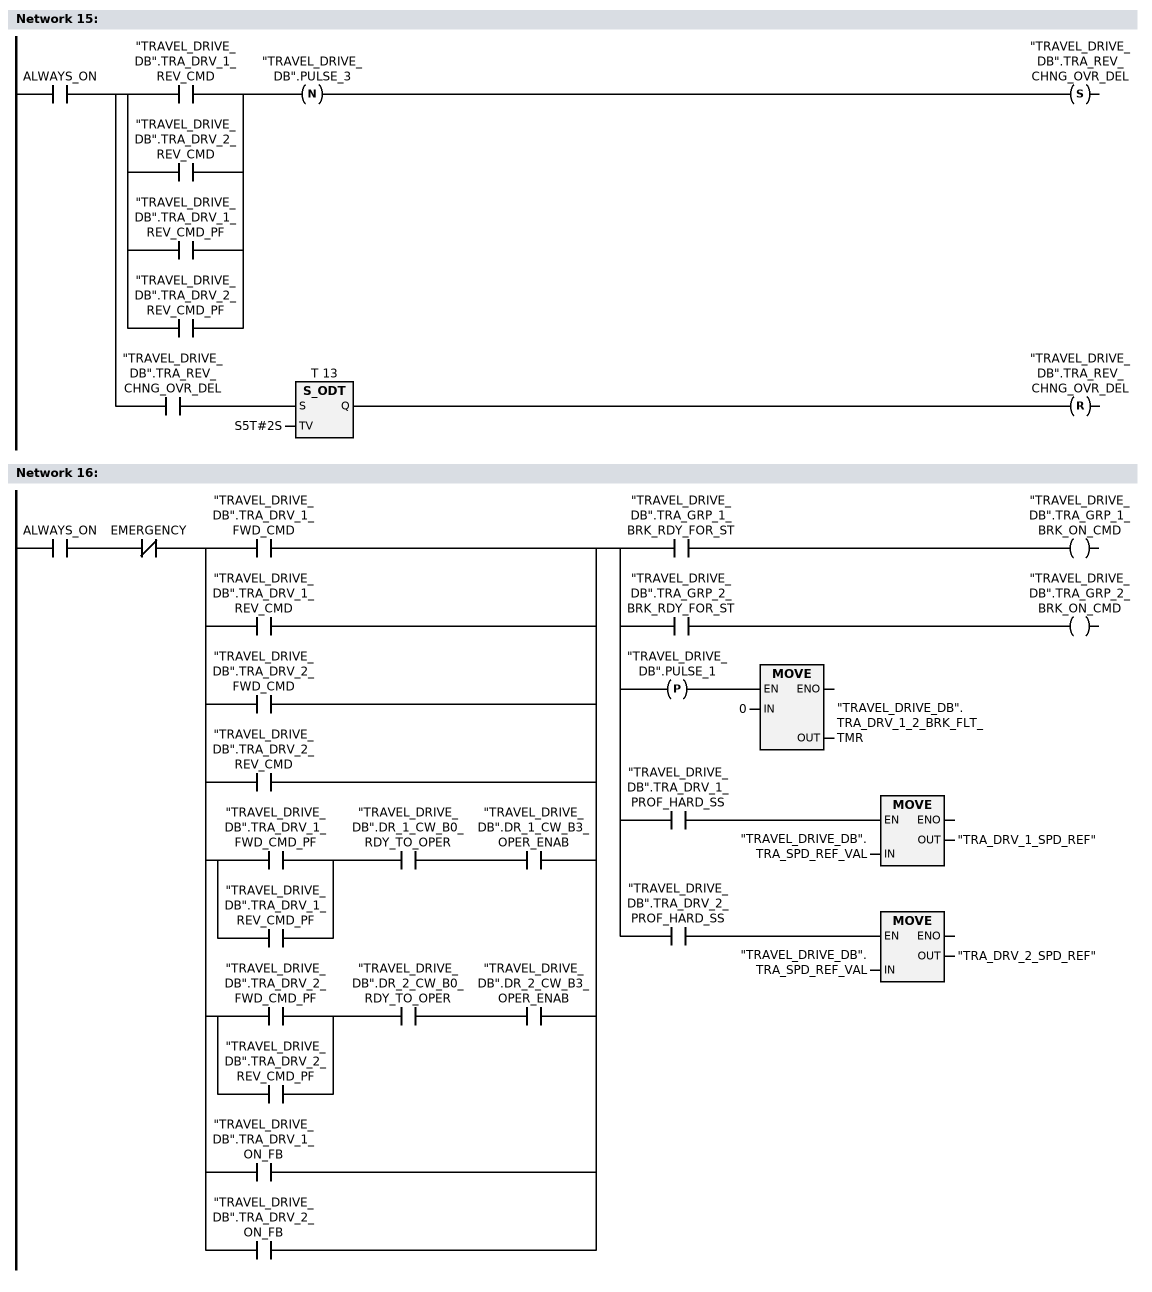
NETWORK
TITLE =
      A     "ALWAYS_ON";
      =     L 0.0;
      A     L 0.0;
      A(;
      O     "TRAVEL_DRIVE_DB".TRA_DRV_1_REV_CMD;
      O     "TRAVEL_DRIVE_DB".TRA_DRV_2_REV_CMD;
      O     "TRAVEL_DRIVE_DB".TRA_DRV_1_REV_CMD_PF;
      O     "TRAVEL_DRIVE_DB".TRA_DRV_2_REV_CMD_PF;
      );
      FN    "TRAVEL_DRIVE_DB".PULSE_3;
      S     "TRAVEL_DRIVE_DB".TRA_REV_CHNG_OVR_DEL;
      A     L 0.0;
      A     "TRAVEL_DRIVE_DB".TRA_REV_CHNG_OVR_DEL;
      L     S5T#2S;
      SD    T 13;
      NOP   0;
      NOP   0;
      NOP   0;
      A     T 13;
      R     "TRAVEL_DRIVE_DB".TRA_REV_CHNG_OVR_DEL;
NETWORK
TITLE =
      A     "ALWAYS_ON";
      AN    "EMERGENCY";
      A(;
      O     "TRAVEL_DRIVE_DB".TRA_DRV_1_FWD_CMD;
      O     "TRAVEL_DRIVE_DB".TRA_DRV_1_REV_CMD;
      O     "TRAVEL_DRIVE_DB".TRA_DRV_2_FWD_CMD;
      O     "TRAVEL_DRIVE_DB".TRA_DRV_2_REV_CMD;
      O;
      A(;
      O     "TRAVEL_DRIVE_DB".TRA_DRV_1_FWD_CMD_PF;
      O     "TRAVEL_DRIVE_DB".TRA_DRV_1_REV_CMD_PF;
      );
      A     "TRAVEL_DRIVE_DB".DR_1_CW_B0_RDY_TO_OPER;
      A     "TRAVEL_DRIVE_DB".DR_1_CW_B3_OPER_ENAB;
      O;
      A(;
      O     "TRAVEL_DRIVE_DB".TRA_DRV_2_FWD_CMD_PF;
      O     "TRAVEL_DRIVE_DB".TRA_DRV_2_REV_CMD_PF;
      );
      A     "TRAVEL_DRIVE_DB".DR_2_CW_B0_RDY_TO_OPER;
      A     "TRAVEL_DRIVE_DB".DR_2_CW_B3_OPER_ENAB;
      O     "TRAVEL_DRIVE_DB".TRA_DRV_1_ON_FB;
      O     "TRAVEL_DRIVE_DB".TRA_DRV_2_ON_FB;
      );
      =     L 0.0;
      A     L 0.0;
      A     "TRAVEL_DRIVE_DB".TRA_GRP_1_BRK_RDY_FOR_ST;
      =     "TRAVEL_DRIVE_DB".TRA_GRP_1_BRK_ON_CMD;
      A     L 0.0;
      A     "TRAVEL_DRIVE_DB".TRA_GRP_2_BRK_RDY_FOR_ST;
      =     "TRAVEL_DRIVE_DB".TRA_GRP_2_BRK_ON_CMD;
      A     L 0.0;
      FP    "TRAVEL_DRIVE_DB".PULSE_1;
      JNB   _00c;
      L     0;
      T     "TRAVEL_DRIVE_DB".TRA_DRV_1_2_BRK_FLT_TMR;
_00c: NOP   0;
      A     L 0.0;
      A     "TRAVEL_DRIVE_DB".TRA_DRV_1_PROF_HARD_SS;
      JNB   _00d;
      L     "TRAVEL_DRIVE_DB".TRA_SPD_REF_VAL;
      T     "TRA_DRV_1_SPD_REF";
_00d: NOP   0;
      A     L 0.0;
      A     "TRAVEL_DRIVE_DB".TRA_DRV_2_PROF_HARD_SS;
      JNB   _00e;
      L     "TRAVEL_DRIVE_DB".TRA_SPD_REF_VAL;
      T     "TRA_DRV_2_SPD_REF";
_00e: NOP   0;
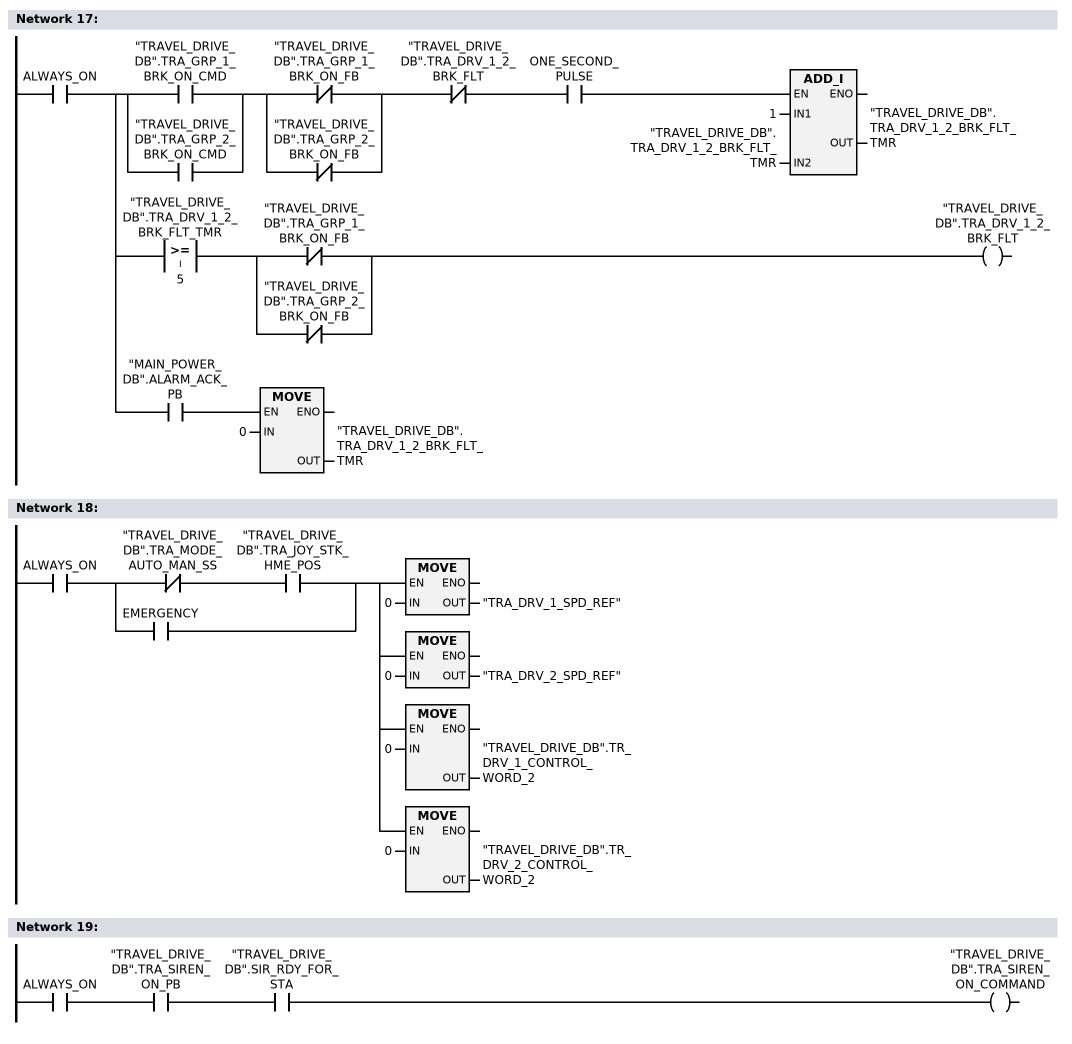
NETWORK
TITLE =
      A     "ALWAYS_ON";
      =     L 0.0;
      A     L 0.0;
      A(;
      O     "TRAVEL_DRIVE_DB".TRA_GRP_1_BRK_ON_CMD;
      O     "TRAVEL_DRIVE_DB".TRA_GRP_2_BRK_ON_CMD;
      );
      A(;
      ON    "TRAVEL_DRIVE_DB".TRA_GRP_1_BRK_ON_FB;
      ON    "TRAVEL_DRIVE_DB".TRA_GRP_2_BRK_ON_FB;
      );
      AN    "TRAVEL_DRIVE_DB".TRA_DRV_1_2_BRK_FLT;
      A     "ONE_SECOND_PULSE";
      JNB   _00f;
      L     1;
      L     "TRAVEL_DRIVE_DB".TRA_DRV_1_2_BRK_FLT_TMR;
      +I;
      T     "TRAVEL_DRIVE_DB".TRA_DRV_1_2_BRK_FLT_TMR;
_00f: NOP   0;
      A     L 0.0;
      A(;
      L     "TRAVEL_DRIVE_DB".TRA_DRV_1_2_BRK_FLT_TMR;
      L     5;
      >=I;
      );
      A(;
      ON    "TRAVEL_DRIVE_DB".TRA_GRP_1_BRK_ON_FB;
      ON    "TRAVEL_DRIVE_DB".TRA_GRP_2_BRK_ON_FB;
      );
      =     "TRAVEL_DRIVE_DB".TRA_DRV_1_2_BRK_FLT;
      A     L 0.0;
      A     "MAIN_POWER_DB".ALARM_ACK_PB;
      JNB   _010;
      L     0;
      T     "TRAVEL_DRIVE_DB".TRA_DRV_1_2_BRK_FLT_TMR;
_010: NOP   0;
NETWORK
TITLE =
      A     "ALWAYS_ON";
      A(;
      AN    "TRAVEL_DRIVE_DB".TRA_MODE_AUTO_MAN_SS;
      A     "TRAVEL_DRIVE_DB".TRA_JOY_STK_HME_POS;
      O     "EMERGENCY";
      );
      =     L 0.0;
      A     L 0.0;
      JNB   _011;
      L     0;
      T     "TRA_DRV_1_SPD_REF";
_011: NOP   0;
      A     L 0.0;
      JNB   _012;
      L     0;
      T     "TRA_DRV_2_SPD_REF";
_012: NOP   0;
      A     L 0.0;
      JNB   _013;
      L     0;
      T     "TRAVEL_DRIVE_DB".TR_DRV_1_CONTROL_WORD_2;
_013: NOP   0;
      A     L 0.0;
      JNB   _014;
      L     0;
      T     "TRAVEL_DRIVE_DB".TR_DRV_2_CONTROL_WORD_2;
_014: NOP   0;
NETWORK
TITLE =
      A     "ALWAYS_ON";
      A     "TRAVEL_DRIVE_DB".TRA_SIREN_ON_PB;
      A     "TRAVEL_DRIVE_DB".SIR_RDY_FOR_STA;
      =     "TRAVEL_DRIVE_DB".TRA_SIREN_ON_COMMAND;
END_FUNCTION

FUNCTION "PUSHER_RAM" : VOID	// FC 8
AUTHOR : Kamillas
VERSION : 0.1
BEGIN
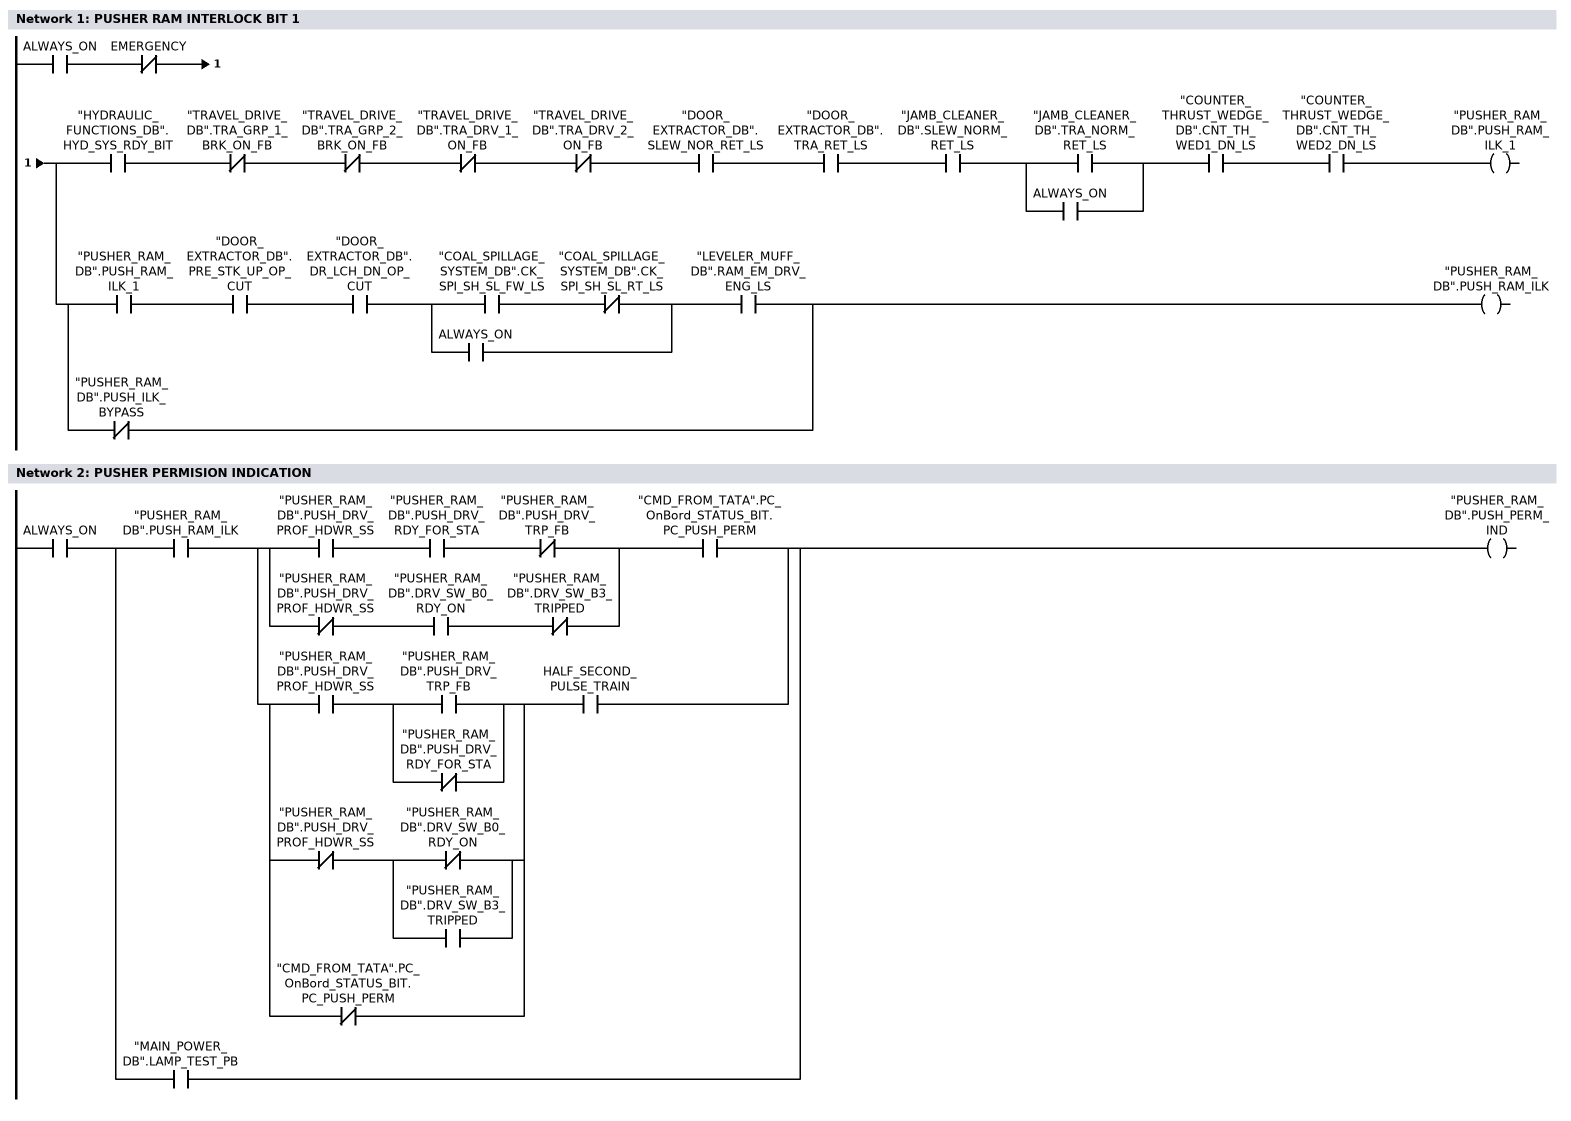
NETWORK
TITLE = PUSHER RAM INTERLOCK BIT 1
      A     "ALWAYS_ON";
      AN    "EMERGENCY";
      =     L 0.0;
      A     L 0.0;
      A     "HYDRAULIC_FUNCTIONS_DB".HYD_SYS_RDY_BIT;
      AN    "TRAVEL_DRIVE_DB".TRA_GRP_1_BRK_ON_FB;
      AN    "TRAVEL_DRIVE_DB".TRA_GRP_2_BRK_ON_FB;
      AN    "TRAVEL_DRIVE_DB".TRA_DRV_1_ON_FB;
      AN    "TRAVEL_DRIVE_DB".TRA_DRV_2_ON_FB;
      A     "DOOR_EXTRACTOR_DB".SLEW_NOR_RET_LS;
      A     "DOOR_EXTRACTOR_DB".TRA_RET_LS;
      A     "JAMB_CLEANER_DB".SLEW_NORM_RET_LS;
      A(;
      O     "JAMB_CLEANER_DB".TRA_NORM_RET_LS;
      O     "ALWAYS_ON";
      );
      A     "COUNTER_THRUST_WEDGE_DB".CNT_TH_WED1_DN_LS;
      A     "COUNTER_THRUST_WEDGE_DB".CNT_TH_WED2_DN_LS;
      =     "PUSHER_RAM_DB".PUSH_RAM_ILK_1;
      A     L 0.0;
      A(;
      A     "PUSHER_RAM_DB".PUSH_RAM_ILK_1;
      A     "DOOR_EXTRACTOR_DB".PRE_STK_UP_OP_CUT;
      A     "DOOR_EXTRACTOR_DB".DR_LCH_DN_OP_CUT;
      A(;
      A     "COAL_SPILLAGE_SYSTEM_DB".CK_SPI_SH_SL_FW_LS;
      AN    "COAL_SPILLAGE_SYSTEM_DB".CK_SPI_SH_SL_RT_LS;
      O     "ALWAYS_ON";
      );
      A     "LEVELER_MUFF_DB".RAM_EM_DRV_ENG_LS;
      ON    "PUSHER_RAM_DB".PUSH_ILK_BYPASS;
      );
      =     "PUSHER_RAM_DB".PUSH_RAM_ILK;
NETWORK
TITLE = PUSHER PERMISION INDICATION
      A     "ALWAYS_ON";
      A(;
      A     "PUSHER_RAM_DB".PUSH_RAM_ILK;
      A(;
      A(;
      A     "PUSHER_RAM_DB".PUSH_DRV_PROF_HDWR_SS;
      A     "PUSHER_RAM_DB".PUSH_DRV_RDY_FOR_STA;
      AN    "PUSHER_RAM_DB".PUSH_DRV_TRP_FB;
      O;
      AN    "PUSHER_RAM_DB".PUSH_DRV_PROF_HDWR_SS;
      A     "PUSHER_RAM_DB".DRV_SW_B0_RDY_ON;
      AN    "PUSHER_RAM_DB".DRV_SW_B3_TRIPPED;
      );
      A     "CMD_FROM_TATA".PC_OnBord_STATUS_BIT.PC_PUSH_PERM;
      O;
      A(;
      A     "PUSHER_RAM_DB".PUSH_DRV_PROF_HDWR_SS;
      A(;
      O     "PUSHER_RAM_DB".PUSH_DRV_TRP_FB;
      ON    "PUSHER_RAM_DB".PUSH_DRV_RDY_FOR_STA;
      );
      O;
      AN    "PUSHER_RAM_DB".PUSH_DRV_PROF_HDWR_SS;
      A(;
      ON    "PUSHER_RAM_DB".DRV_SW_B0_RDY_ON;
      O     "PUSHER_RAM_DB".DRV_SW_B3_TRIPPED;
      );
      ON    "CMD_FROM_TATA".PC_OnBord_STATUS_BIT.PC_PUSH_PERM;
      );
      A     "HALF_SECOND_PULSE_TRAIN";
      );
      O     "MAIN_POWER_DB".LAMP_TEST_PB;
      );
      =     "PUSHER_RAM_DB".PUSH_PERM_IND;
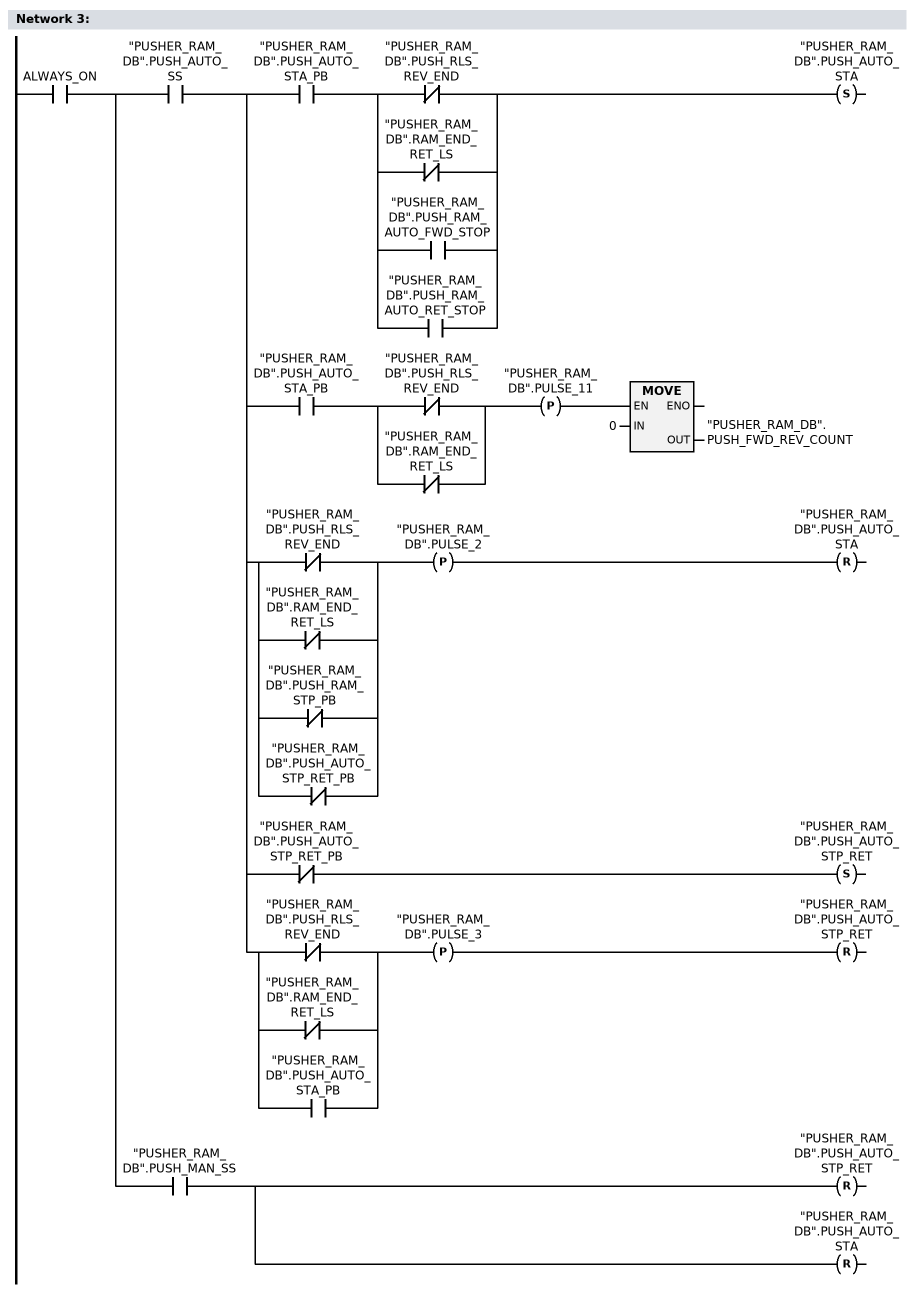
NETWORK
TITLE =
      A     "ALWAYS_ON";
      =     L 0.0;
      A     L 0.0;
      A     "PUSHER_RAM_DB".PUSH_AUTO_SS;
      =     L 0.1;
      A     L 0.1;
      A     "PUSHER_RAM_DB".PUSH_AUTO_STA_PB;
      A(;
      ON    "PUSHER_RAM_DB".PUSH_RLS_REV_END;
      ON    "PUSHER_RAM_DB".RAM_END_RET_LS;
      O     "PUSHER_RAM_DB".PUSH_RAM_AUTO_FWD_STOP;
      O     "PUSHER_RAM_DB".PUSH_RAM_AUTO_RET_STOP;
      );
      S     "PUSHER_RAM_DB".PUSH_AUTO_STA;
      A     L 0.1;
      A     "PUSHER_RAM_DB".PUSH_AUTO_STA_PB;
      A(;
      ON    "PUSHER_RAM_DB".PUSH_RLS_REV_END;
      ON    "PUSHER_RAM_DB".RAM_END_RET_LS;
      );
      FP    "PUSHER_RAM_DB".PULSE_11;
      JNB   _001;
      L     0;
      T     "PUSHER_RAM_DB".PUSH_FWD_REV_COUNT;
_001: NOP   0;
      A     L 0.1;
      A(;
      ON    "PUSHER_RAM_DB".PUSH_RLS_REV_END;
      ON    "PUSHER_RAM_DB".RAM_END_RET_LS;
      ON    "PUSHER_RAM_DB".PUSH_RAM_STP_PB;
      ON    "PUSHER_RAM_DB".PUSH_AUTO_STP_RET_PB;
      );
      FP    "PUSHER_RAM_DB".PULSE_2;
      R     "PUSHER_RAM_DB".PUSH_AUTO_STA;
      A     L 0.1;
      AN    "PUSHER_RAM_DB".PUSH_AUTO_STP_RET_PB;
      S     "PUSHER_RAM_DB".PUSH_AUTO_STP_RET;
      A     L 0.1;
      A(;
      ON    "PUSHER_RAM_DB".PUSH_RLS_REV_END;
      ON    "PUSHER_RAM_DB".RAM_END_RET_LS;
      O     "PUSHER_RAM_DB".PUSH_AUTO_STA_PB;
      );
      FP    "PUSHER_RAM_DB".PULSE_3;
      R     "PUSHER_RAM_DB".PUSH_AUTO_STP_RET;
      A     L 0.0;
      A     "PUSHER_RAM_DB".PUSH_MAN_SS;
      R     "PUSHER_RAM_DB".PUSH_AUTO_STP_RET;
      R     "PUSHER_RAM_DB".PUSH_AUTO_STA;
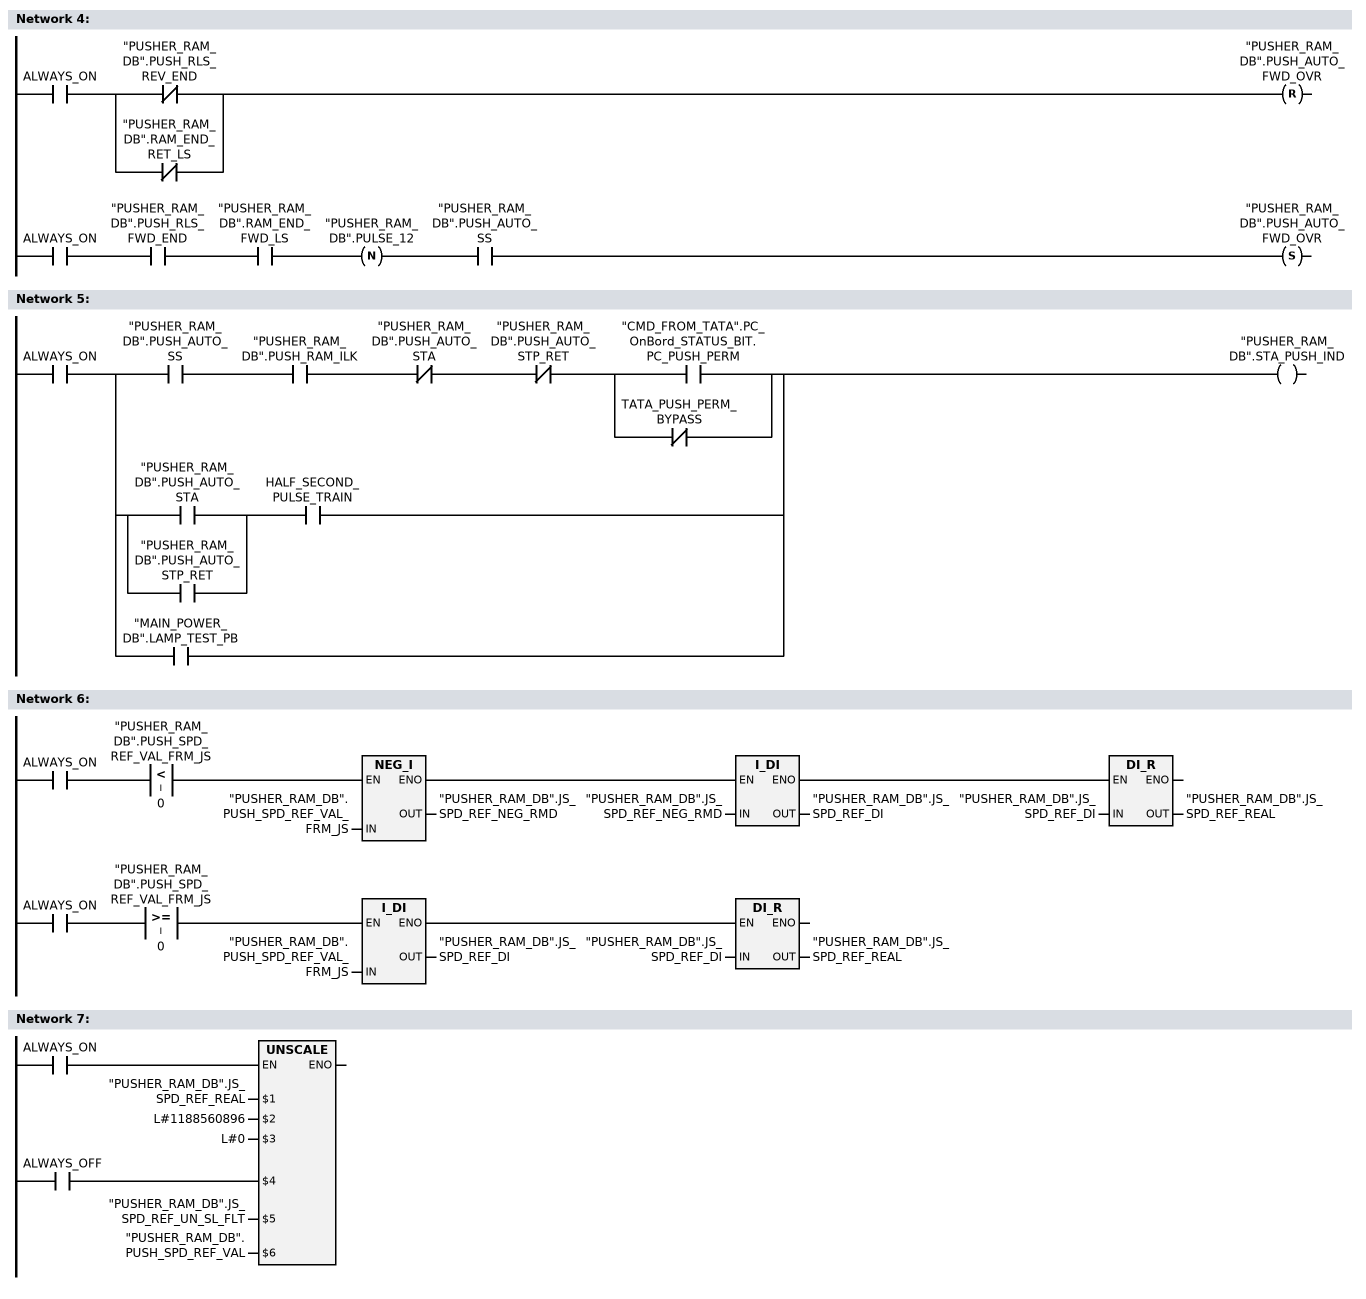
NETWORK
TITLE =
      A     "ALWAYS_ON";
      =     L 0.0;
      A(;
      A     L 0.0;
      A     "PUSHER_RAM_DB".PUSH_RLS_FWD_END;
      A     "PUSHER_RAM_DB".RAM_END_FWD_LS;
      FN    "PUSHER_RAM_DB".PULSE_12;
      );
      A     "PUSHER_RAM_DB".PUSH_AUTO_SS;
      S     "PUSHER_RAM_DB".PUSH_AUTO_FWD_OVR;
      A     L 0.0;
      A(;
      ON    "PUSHER_RAM_DB".PUSH_RLS_REV_END;
      ON    "PUSHER_RAM_DB".RAM_END_RET_LS;
      );
      R     "PUSHER_RAM_DB".PUSH_AUTO_FWD_OVR;
NETWORK
TITLE =
      A     "ALWAYS_ON";
      A(;
      A     "PUSHER_RAM_DB".PUSH_AUTO_SS;
      A     "PUSHER_RAM_DB".PUSH_RAM_ILK;
      AN    "PUSHER_RAM_DB".PUSH_AUTO_STA;
      AN    "PUSHER_RAM_DB".PUSH_AUTO_STP_RET;
      A(;
      O     "CMD_FROM_TATA".PC_OnBord_STATUS_BIT.PC_PUSH_PERM;
      ON    "TATA_PUSH_PERM_BYPASS";
      );
      O;
      A(;
      O     "PUSHER_RAM_DB".PUSH_AUTO_STA;
      O     "PUSHER_RAM_DB".PUSH_AUTO_STP_RET;
      );
      A     "HALF_SECOND_PULSE_TRAIN";
      O     "MAIN_POWER_DB".LAMP_TEST_PB;
      );
      =     "PUSHER_RAM_DB".STA_PUSH_IND;
NETWORK
TITLE =
      A     "ALWAYS_ON";
      =     L 0.0;
      A(;
      A(;
      A     L 0.0;
      A(;
      L     "PUSHER_RAM_DB".PUSH_SPD_REF_VAL_FRM_JS;
      L     0;
      <I;
      );
      JNB   _002;
      L     "PUSHER_RAM_DB".PUSH_SPD_REF_VAL_FRM_JS;
      NEGI;
      T     "PUSHER_RAM_DB".JS_SPD_REF_NEG_RMD;
      AN    OV;
      SAVE;
      CLR;
_002: A     BR;
      );
      JNB   _003;
      L     "PUSHER_RAM_DB".JS_SPD_REF_NEG_RMD;
      ITD;
      T     "PUSHER_RAM_DB".JS_SPD_REF_DI;
      SET;
      SAVE;
      CLR;
_003: A     BR;
      );
      JNB   _004;
      L     "PUSHER_RAM_DB".JS_SPD_REF_DI;
      DTR;
      T     "PUSHER_RAM_DB".JS_SPD_REF_REAL;
_004: NOP   0;
      A(;
      A     L 0.0;
      A(;
      L     "PUSHER_RAM_DB".PUSH_SPD_REF_VAL_FRM_JS;
      L     0;
      >=I;
      );
      JNB   _005;
      L     "PUSHER_RAM_DB".PUSH_SPD_REF_VAL_FRM_JS;
      ITD;
      T     "PUSHER_RAM_DB".JS_SPD_REF_DI;
      SET;
      SAVE;
      CLR;
_005: A     BR;
      );
      JNB   _006;
      L     "PUSHER_RAM_DB".JS_SPD_REF_DI;
      DTR;
      T     "PUSHER_RAM_DB".JS_SPD_REF_REAL;
_006: NOP   0;
NETWORK
TITLE =
      A     "ALWAYS_OFF";
      =     L 0.0;
      BLD   103;
      A     "ALWAYS_ON";
      JNB   _007;
      CALL  "UNSCALE" (
           $1                       := "PUSHER_RAM_DB".JS_SPD_REF_REAL,
           $2                       := L#1188560896,
           $3                       := L#0,
           $4                       := L 0.0,
           $5                       := "PUSHER_RAM_DB".JS_SPD_REF_UN_SL_FLT,
           $6                       := "PUSHER_RAM_DB".PUSH_SPD_REF_VAL);
_007: NOP   0;
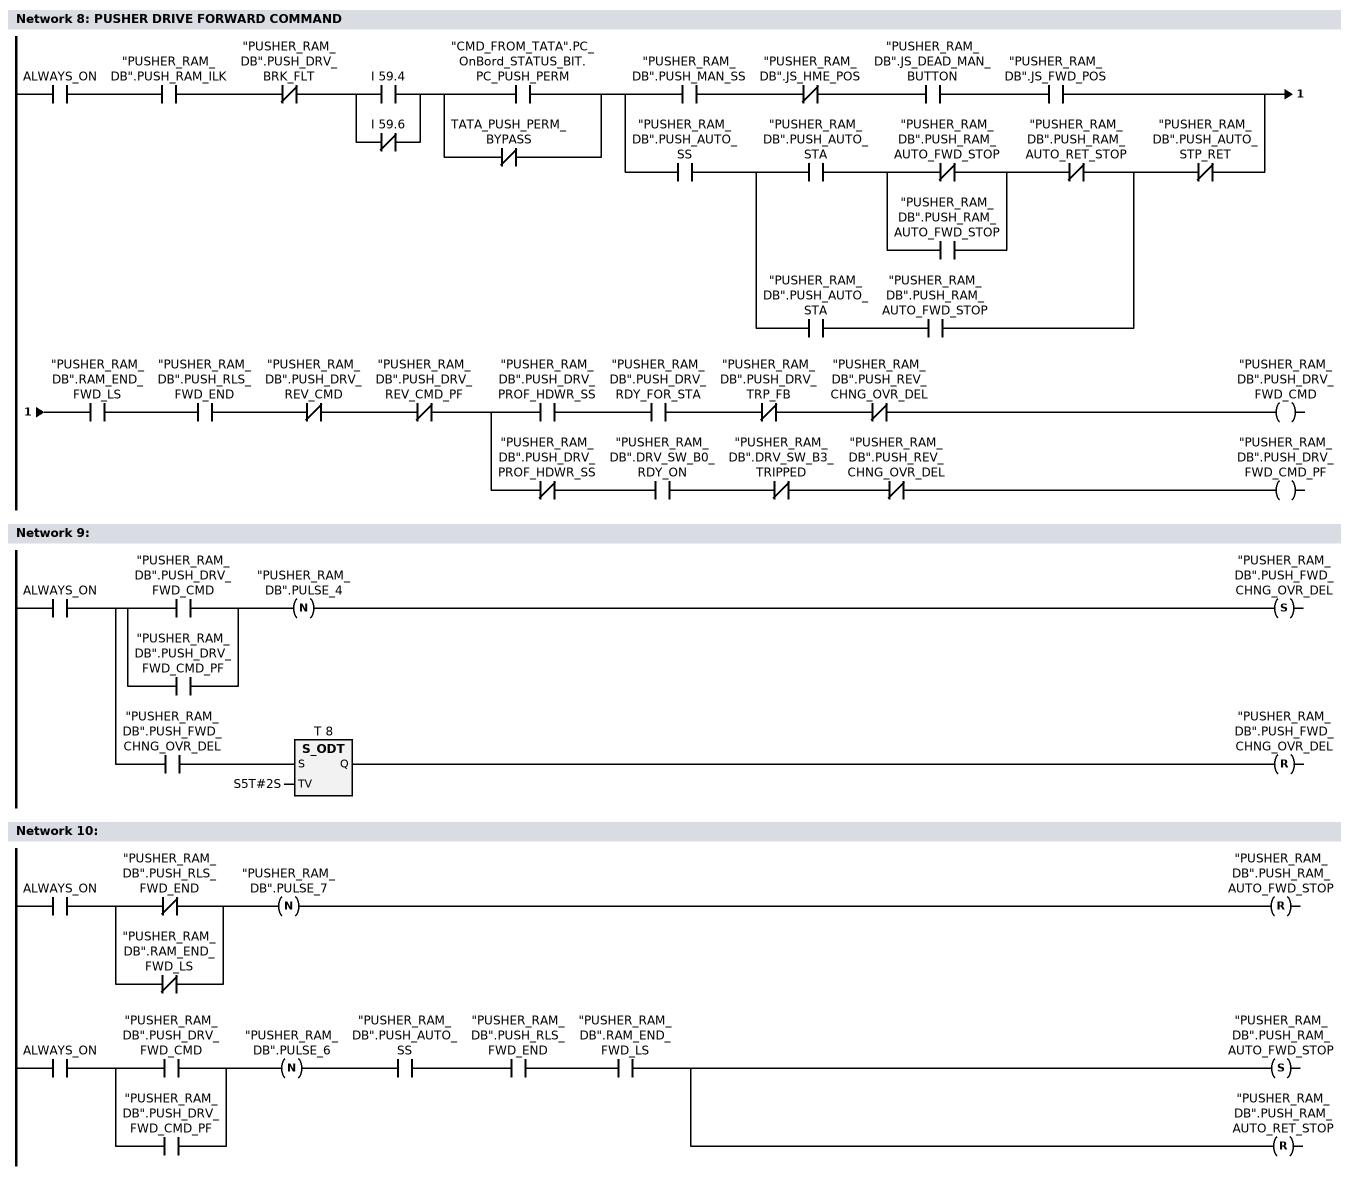
NETWORK
TITLE = PUSHER DRIVE FORWARD COMMAND
      A     "ALWAYS_ON";
      A     "PUSHER_RAM_DB".PUSH_RAM_ILK;
      AN    "PUSHER_RAM_DB".PUSH_DRV_BRK_FLT;
      A(;
      O     I 59.4;
      ON    I 59.6;
      );
      A(;
      O     "CMD_FROM_TATA".PC_OnBord_STATUS_BIT.PC_PUSH_PERM;
      ON    "TATA_PUSH_PERM_BYPASS";
      );
      A(;
      A     "PUSHER_RAM_DB".PUSH_MAN_SS;
      AN    "PUSHER_RAM_DB".JS_HME_POS;
      A     "PUSHER_RAM_DB".JS_DEAD_MAN_BUTTON;
      A     "PUSHER_RAM_DB".JS_FWD_POS;
      O;
      A     "PUSHER_RAM_DB".PUSH_AUTO_SS;
      A(;
      A     "PUSHER_RAM_DB".PUSH_AUTO_STA;
      A(;
      ON    "PUSHER_RAM_DB".PUSH_RAM_AUTO_FWD_STOP;
      O     "PUSHER_RAM_DB".PUSH_RAM_AUTO_FWD_STOP;
      );
      AN    "PUSHER_RAM_DB".PUSH_RAM_AUTO_RET_STOP;
      O;
      A     "PUSHER_RAM_DB".PUSH_AUTO_STA;
      A     "PUSHER_RAM_DB".PUSH_RAM_AUTO_FWD_STOP;
      );
      AN    "PUSHER_RAM_DB".PUSH_AUTO_STP_RET;
      );
      A     "PUSHER_RAM_DB".RAM_END_FWD_LS;
      A     "PUSHER_RAM_DB".PUSH_RLS_FWD_END;
      AN    "PUSHER_RAM_DB".PUSH_DRV_REV_CMD;
      AN    "PUSHER_RAM_DB".PUSH_DRV_REV_CMD_PF;
      =     L 0.0;
      A     L 0.0;
      A     "PUSHER_RAM_DB".PUSH_DRV_PROF_HDWR_SS;
      A     "PUSHER_RAM_DB".PUSH_DRV_RDY_FOR_STA;
      AN    "PUSHER_RAM_DB".PUSH_DRV_TRP_FB;
      AN    "PUSHER_RAM_DB".PUSH_REV_CHNG_OVR_DEL;
      =     "PUSHER_RAM_DB".PUSH_DRV_FWD_CMD;
      A     L 0.0;
      AN    "PUSHER_RAM_DB".PUSH_DRV_PROF_HDWR_SS;
      A     "PUSHER_RAM_DB".DRV_SW_B0_RDY_ON;
      AN    "PUSHER_RAM_DB".DRV_SW_B3_TRIPPED;
      AN    "PUSHER_RAM_DB".PUSH_REV_CHNG_OVR_DEL;
      =     "PUSHER_RAM_DB".PUSH_DRV_FWD_CMD_PF;
NETWORK
TITLE =
      A     "ALWAYS_ON";
      =     L 0.0;
      A     L 0.0;
      A(;
      O     "PUSHER_RAM_DB".PUSH_DRV_FWD_CMD;
      O     "PUSHER_RAM_DB".PUSH_DRV_FWD_CMD_PF;
      );
      FN    "PUSHER_RAM_DB".PULSE_4;
      S     "PUSHER_RAM_DB".PUSH_FWD_CHNG_OVR_DEL;
      A     L 0.0;
      A     "PUSHER_RAM_DB".PUSH_FWD_CHNG_OVR_DEL;
      L     S5T#2S;
      SD    T 8;
      NOP   0;
      NOP   0;
      NOP   0;
      A     T 8;
      R     "PUSHER_RAM_DB".PUSH_FWD_CHNG_OVR_DEL;
NETWORK
TITLE =
      A     "ALWAYS_ON";
      =     L 0.0;
      A(;
      A     L 0.0;
      A(;
      O     "PUSHER_RAM_DB".PUSH_DRV_FWD_CMD;
      O     "PUSHER_RAM_DB".PUSH_DRV_FWD_CMD_PF;
      );
      FN    "PUSHER_RAM_DB".PULSE_6;
      );
      A     "PUSHER_RAM_DB".PUSH_AUTO_SS;
      A     "PUSHER_RAM_DB".PUSH_RLS_FWD_END;
      A     "PUSHER_RAM_DB".RAM_END_FWD_LS;
      S     "PUSHER_RAM_DB".PUSH_RAM_AUTO_FWD_STOP;
      R     "PUSHER_RAM_DB".PUSH_RAM_AUTO_RET_STOP;
      A     L 0.0;
      A(;
      ON    "PUSHER_RAM_DB".PUSH_RLS_FWD_END;
      ON    "PUSHER_RAM_DB".RAM_END_FWD_LS;
      );
      FN    "PUSHER_RAM_DB".PULSE_7;
      R     "PUSHER_RAM_DB".PUSH_RAM_AUTO_FWD_STOP;
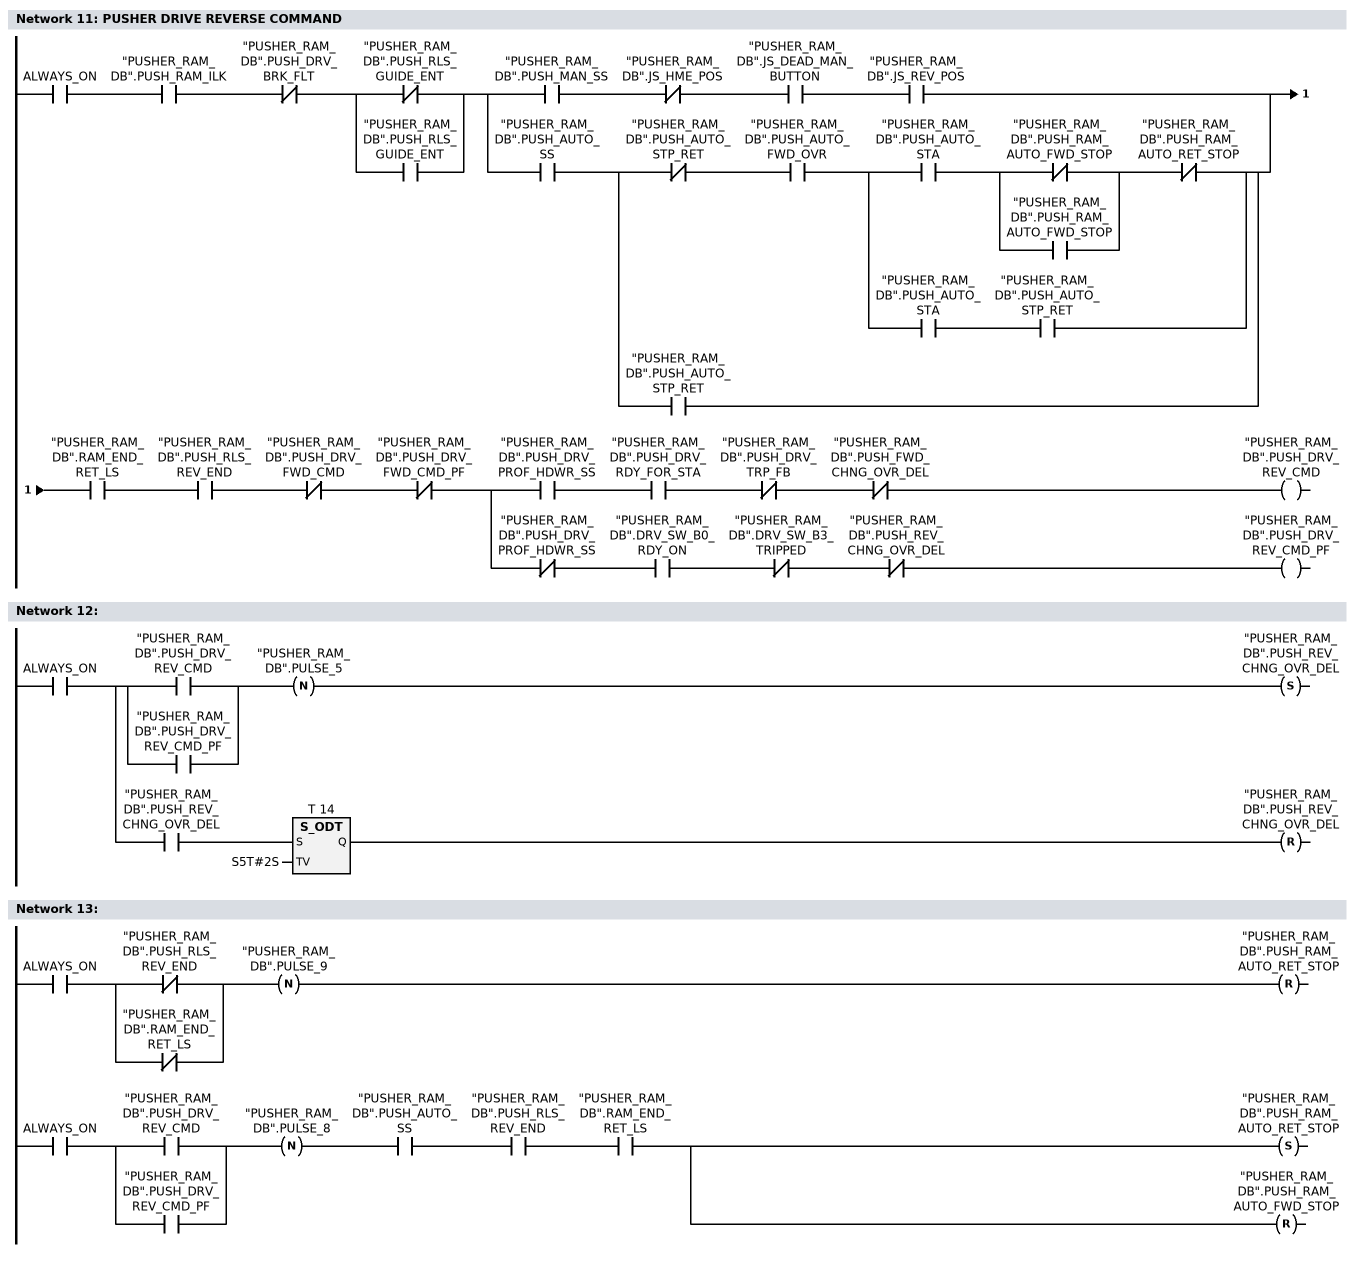
NETWORK
TITLE = PUSHER DRIVE REVERSE COMMAND
      A     "ALWAYS_ON";
      A     "PUSHER_RAM_DB".PUSH_RAM_ILK;
      AN    "PUSHER_RAM_DB".PUSH_DRV_BRK_FLT;
      A(;
      ON    "PUSHER_RAM_DB".PUSH_RLS_GUIDE_ENT;
      O     "PUSHER_RAM_DB".PUSH_RLS_GUIDE_ENT;
      );
      A(;
      A     "PUSHER_RAM_DB".PUSH_MAN_SS;
      AN    "PUSHER_RAM_DB".JS_HME_POS;
      A     "PUSHER_RAM_DB".JS_DEAD_MAN_BUTTON;
      A     "PUSHER_RAM_DB".JS_REV_POS;
      O;
      A     "PUSHER_RAM_DB".PUSH_AUTO_SS;
      A(;
      AN    "PUSHER_RAM_DB".PUSH_AUTO_STP_RET;
      A     "PUSHER_RAM_DB".PUSH_AUTO_FWD_OVR;
      A(;
      A     "PUSHER_RAM_DB".PUSH_AUTO_STA;
      A(;
      ON    "PUSHER_RAM_DB".PUSH_RAM_AUTO_FWD_STOP;
      O     "PUSHER_RAM_DB".PUSH_RAM_AUTO_FWD_STOP;
      );
      AN    "PUSHER_RAM_DB".PUSH_RAM_AUTO_RET_STOP;
      O;
      A     "PUSHER_RAM_DB".PUSH_AUTO_STA;
      A     "PUSHER_RAM_DB".PUSH_AUTO_STP_RET;
      );
      O     "PUSHER_RAM_DB".PUSH_AUTO_STP_RET;
      );
      );
      A     "PUSHER_RAM_DB".RAM_END_RET_LS;
      A     "PUSHER_RAM_DB".PUSH_RLS_REV_END;
      AN    "PUSHER_RAM_DB".PUSH_DRV_FWD_CMD;
      AN    "PUSHER_RAM_DB".PUSH_DRV_FWD_CMD_PF;
      =     L 0.0;
      A     L 0.0;
      A     "PUSHER_RAM_DB".PUSH_DRV_PROF_HDWR_SS;
      A     "PUSHER_RAM_DB".PUSH_DRV_RDY_FOR_STA;
      AN    "PUSHER_RAM_DB".PUSH_DRV_TRP_FB;
      AN    "PUSHER_RAM_DB".PUSH_FWD_CHNG_OVR_DEL;
      =     "PUSHER_RAM_DB".PUSH_DRV_REV_CMD;
      A     L 0.0;
      AN    "PUSHER_RAM_DB".PUSH_DRV_PROF_HDWR_SS;
      A     "PUSHER_RAM_DB".DRV_SW_B0_RDY_ON;
      AN    "PUSHER_RAM_DB".DRV_SW_B3_TRIPPED;
      AN    "PUSHER_RAM_DB".PUSH_REV_CHNG_OVR_DEL;
      =     "PUSHER_RAM_DB".PUSH_DRV_REV_CMD_PF;
NETWORK
TITLE =
      A     "ALWAYS_ON";
      =     L 0.0;
      A     L 0.0;
      A(;
      O     "PUSHER_RAM_DB".PUSH_DRV_REV_CMD;
      O     "PUSHER_RAM_DB".PUSH_DRV_REV_CMD_PF;
      );
      FN    "PUSHER_RAM_DB".PULSE_5;
      S     "PUSHER_RAM_DB".PUSH_REV_CHNG_OVR_DEL;
      A     L 0.0;
      A     "PUSHER_RAM_DB".PUSH_REV_CHNG_OVR_DEL;
      L     S5T#2S;
      SD    T 14;
      NOP   0;
      NOP   0;
      NOP   0;
      A     T 14;
      R     "PUSHER_RAM_DB".PUSH_REV_CHNG_OVR_DEL;
NETWORK
TITLE =
      A     "ALWAYS_ON";
      =     L 0.0;
      A(;
      A     L 0.0;
      A(;
      O     "PUSHER_RAM_DB".PUSH_DRV_REV_CMD;
      O     "PUSHER_RAM_DB".PUSH_DRV_REV_CMD_PF;
      );
      FN    "PUSHER_RAM_DB".PULSE_8;
      );
      A     "PUSHER_RAM_DB".PUSH_AUTO_SS;
      A     "PUSHER_RAM_DB".PUSH_RLS_REV_END;
      A     "PUSHER_RAM_DB".RAM_END_RET_LS;
      S     "PUSHER_RAM_DB".PUSH_RAM_AUTO_RET_STOP;
      R     "PUSHER_RAM_DB".PUSH_RAM_AUTO_FWD_STOP;
      A     L 0.0;
      A(;
      ON    "PUSHER_RAM_DB".PUSH_RLS_REV_END;
      ON    "PUSHER_RAM_DB".RAM_END_RET_LS;
      );
      FN    "PUSHER_RAM_DB".PULSE_9;
      R     "PUSHER_RAM_DB".PUSH_RAM_AUTO_RET_STOP;
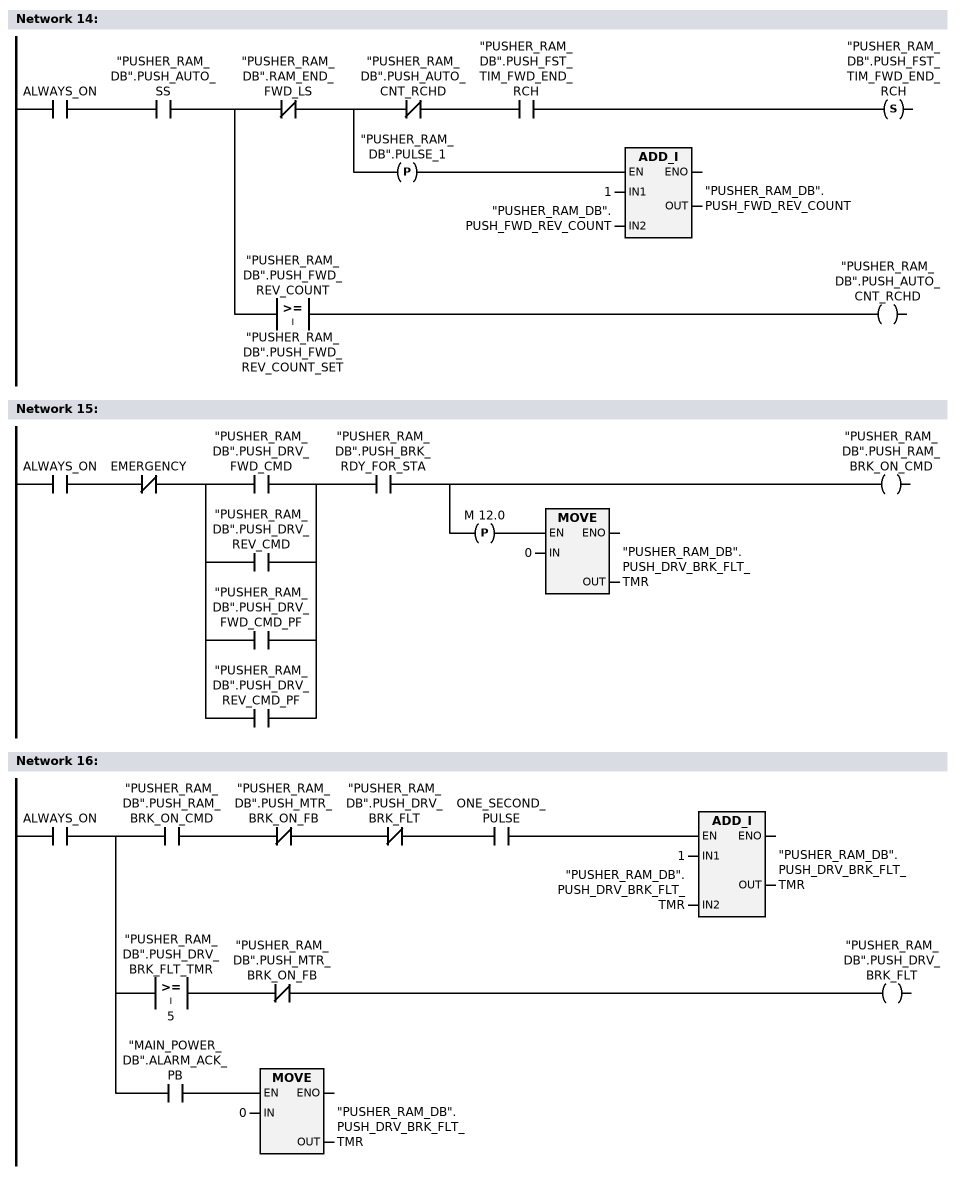
NETWORK
TITLE =
      A     "ALWAYS_ON";
      A     "PUSHER_RAM_DB".PUSH_AUTO_SS;
      =     L 0.0;
      A     L 0.0;
      AN    "PUSHER_RAM_DB".RAM_END_FWD_LS;
      =     L 0.1;
      A     L 0.1;
      AN    "PUSHER_RAM_DB".PUSH_AUTO_CNT_RCHD;
      A     "PUSHER_RAM_DB".PUSH_FST_TIM_FWD_END_RCH;
      S     "PUSHER_RAM_DB".PUSH_FST_TIM_FWD_END_RCH;
      A     L 0.1;
      FP    "PUSHER_RAM_DB".PULSE_1;
      JNB   _008;
      L     1;
      L     "PUSHER_RAM_DB".PUSH_FWD_REV_COUNT;
      +I;
      T     "PUSHER_RAM_DB".PUSH_FWD_REV_COUNT;
_008: NOP   0;
      A     L 0.0;
      A(;
      L     "PUSHER_RAM_DB".PUSH_FWD_REV_COUNT;
      L     "PUSHER_RAM_DB".PUSH_FWD_REV_COUNT_SET;
      >=I;
      );
      =     "PUSHER_RAM_DB".PUSH_AUTO_CNT_RCHD;
NETWORK
TITLE =
      A     "ALWAYS_ON";
      AN    "EMERGENCY";
      A(;
      O     "PUSHER_RAM_DB".PUSH_DRV_FWD_CMD;
      O     "PUSHER_RAM_DB".PUSH_DRV_REV_CMD;
      O     "PUSHER_RAM_DB".PUSH_DRV_FWD_CMD_PF;
      O     "PUSHER_RAM_DB".PUSH_DRV_REV_CMD_PF;
      );
      A     "PUSHER_RAM_DB".PUSH_BRK_RDY_FOR_STA;
      =     L 0.0;
      A     L 0.0;
      BLD   102;
      =     "PUSHER_RAM_DB".PUSH_RAM_BRK_ON_CMD;
      A     L 0.0;
      FP    M 12.0;
      JNB   _009;
      L     0;
      T     "PUSHER_RAM_DB".PUSH_DRV_BRK_FLT_TMR;
_009: NOP   0;
NETWORK
TITLE =
      A     "ALWAYS_ON";
      =     L 0.0;
      A     L 0.0;
      A     "PUSHER_RAM_DB".PUSH_RAM_BRK_ON_CMD;
      AN    "PUSHER_RAM_DB".PUSH_MTR_BRK_ON_FB;
      AN    "PUSHER_RAM_DB".PUSH_DRV_BRK_FLT;
      A     "ONE_SECOND_PULSE";
      JNB   _00a;
      L     1;
      L     "PUSHER_RAM_DB".PUSH_DRV_BRK_FLT_TMR;
      +I;
      T     "PUSHER_RAM_DB".PUSH_DRV_BRK_FLT_TMR;
_00a: NOP   0;
      A     L 0.0;
      A(;
      L     "PUSHER_RAM_DB".PUSH_DRV_BRK_FLT_TMR;
      L     5;
      >=I;
      );
      AN    "PUSHER_RAM_DB".PUSH_MTR_BRK_ON_FB;
      =     "PUSHER_RAM_DB".PUSH_DRV_BRK_FLT;
      A     L 0.0;
      A     "MAIN_POWER_DB".ALARM_ACK_PB;
      JNB   _00b;
      L     0;
      T     "PUSHER_RAM_DB".PUSH_DRV_BRK_FLT_TMR;
_00b: NOP   0;
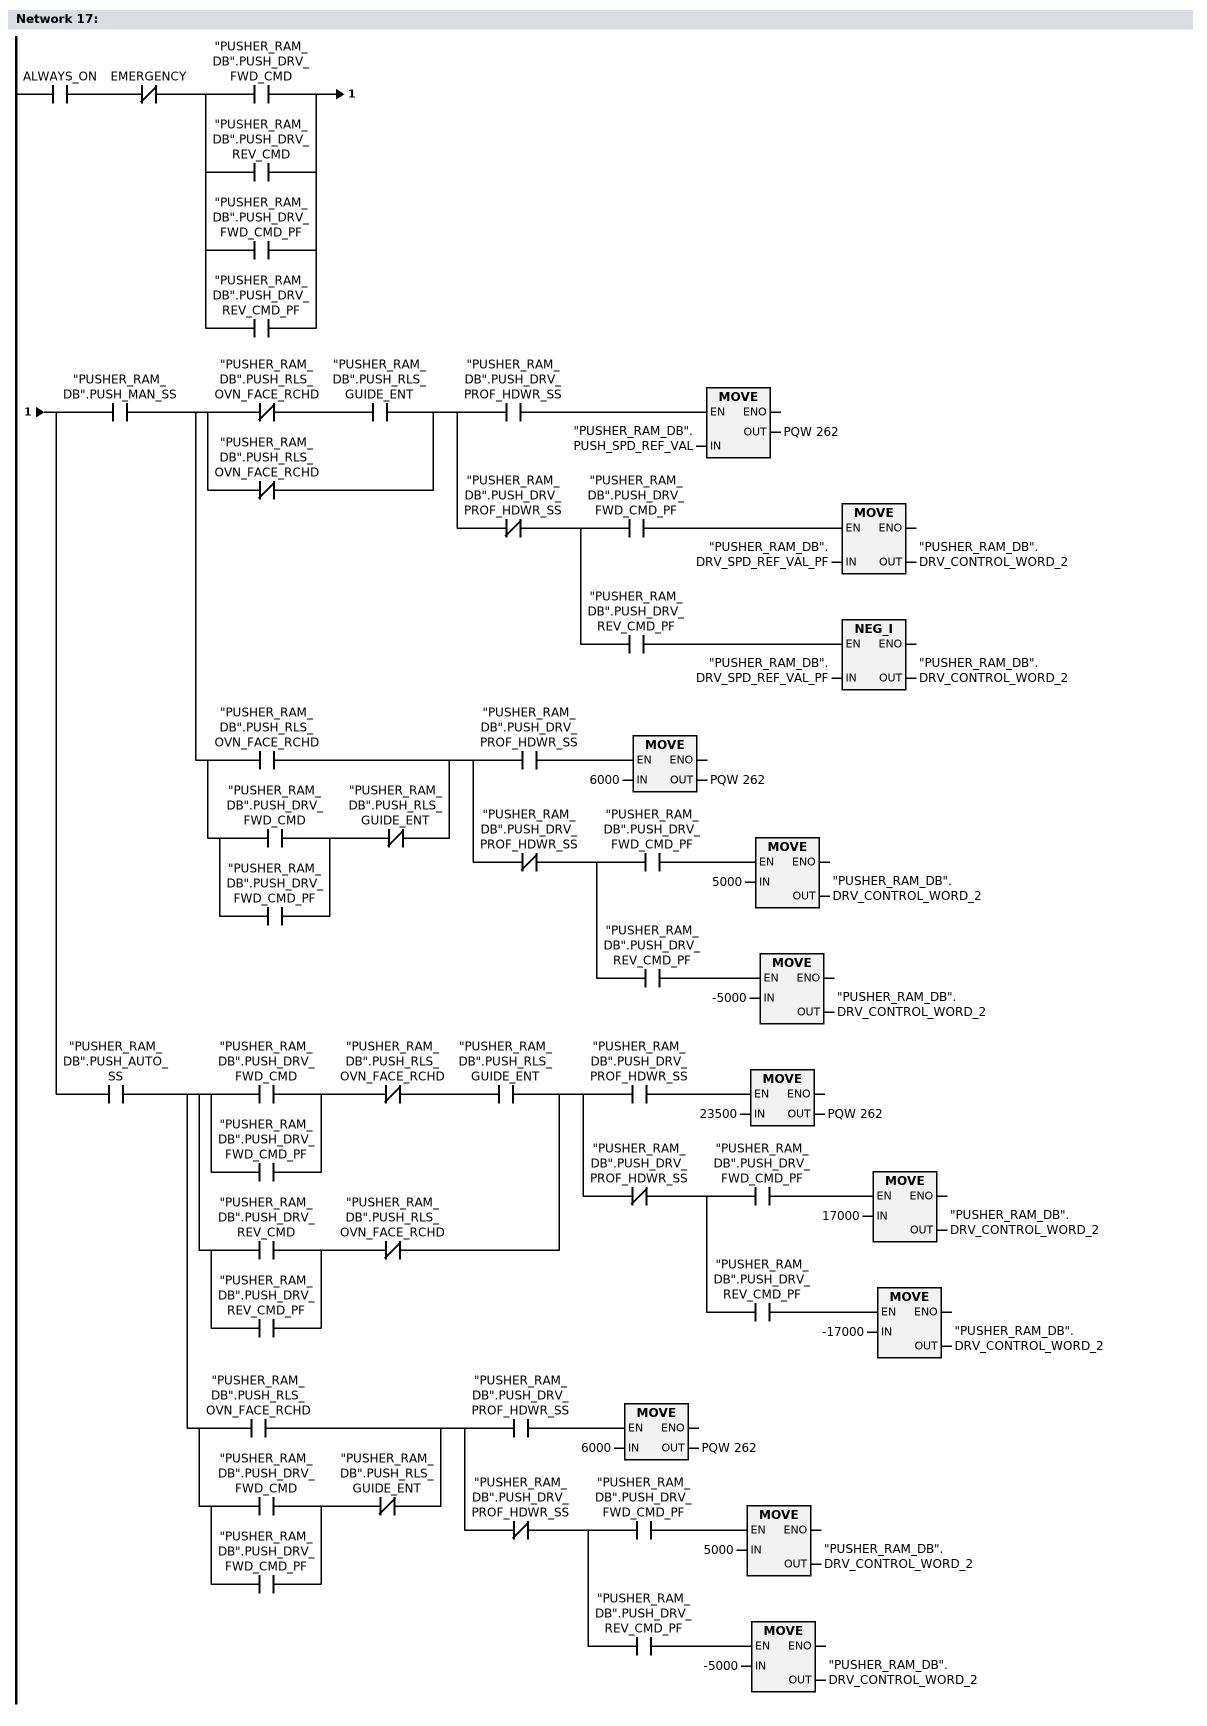
NETWORK
TITLE =
      A     "ALWAYS_ON";
      AN    "EMERGENCY";
      A(;
      O     "PUSHER_RAM_DB".PUSH_DRV_FWD_CMD;
      O     "PUSHER_RAM_DB".PUSH_DRV_REV_CMD;
      O     "PUSHER_RAM_DB".PUSH_DRV_FWD_CMD_PF;
      O     "PUSHER_RAM_DB".PUSH_DRV_REV_CMD_PF;
      );
      =     L 0.0;
      A     L 0.0;
      A     "PUSHER_RAM_DB".PUSH_MAN_SS;
      =     L 0.1;
      A     L 0.1;
      A(;
      AN    "PUSHER_RAM_DB".PUSH_RLS_OVN_FACE_RCHD;
      A     "PUSHER_RAM_DB".PUSH_RLS_GUIDE_ENT;
      ON    "PUSHER_RAM_DB".PUSH_RLS_OVN_FACE_RCHD;
      );
      =     L 0.2;
      A     L 0.2;
      A     "PUSHER_RAM_DB".PUSH_DRV_PROF_HDWR_SS;
      JNB   _00c;
      L     "PUSHER_RAM_DB".PUSH_SPD_REF_VAL;
      T     PQW 262;
_00c: NOP   0;
      A     L 0.2;
      AN    "PUSHER_RAM_DB".PUSH_DRV_PROF_HDWR_SS;
      =     L 0.3;
      A     L 0.3;
      A     "PUSHER_RAM_DB".PUSH_DRV_FWD_CMD_PF;
      JNB   _00d;
      L     "PUSHER_RAM_DB".DRV_SPD_REF_VAL_PF;
      T     "PUSHER_RAM_DB".DRV_CONTROL_WORD_2;
_00d: NOP   0;
      A     L 0.3;
      A     "PUSHER_RAM_DB".PUSH_DRV_REV_CMD_PF;
      JNB   _00e;
      L     "PUSHER_RAM_DB".DRV_SPD_REF_VAL_PF;
      NEGI;
      T     "PUSHER_RAM_DB".DRV_CONTROL_WORD_2;
_00e: NOP   0;
      A     L 0.1;
      A(;
      O     "PUSHER_RAM_DB".PUSH_RLS_OVN_FACE_RCHD;
      O;
      A(;
      O     "PUSHER_RAM_DB".PUSH_DRV_FWD_CMD;
      O     "PUSHER_RAM_DB".PUSH_DRV_FWD_CMD_PF;
      );
      AN    "PUSHER_RAM_DB".PUSH_RLS_GUIDE_ENT;
      );
      =     L 0.2;
      A     L 0.2;
      A     "PUSHER_RAM_DB".PUSH_DRV_PROF_HDWR_SS;
      JNB   _00f;
      L     6000;
      T     PQW 262;
_00f: NOP   0;
      A     L 0.2;
      AN    "PUSHER_RAM_DB".PUSH_DRV_PROF_HDWR_SS;
      =     L 0.3;
      A     L 0.3;
      A     "PUSHER_RAM_DB".PUSH_DRV_FWD_CMD_PF;
      JNB   _010;
      L     5000;
      T     "PUSHER_RAM_DB".DRV_CONTROL_WORD_2;
_010: NOP   0;
      A     L 0.3;
      A     "PUSHER_RAM_DB".PUSH_DRV_REV_CMD_PF;
      JNB   _011;
      L     -5000;
      T     "PUSHER_RAM_DB".DRV_CONTROL_WORD_2;
_011: NOP   0;
      A     L 0.0;
      A     "PUSHER_RAM_DB".PUSH_AUTO_SS;
      =     L 0.1;
      A     L 0.1;
      A(;
      A(;
      O     "PUSHER_RAM_DB".PUSH_DRV_FWD_CMD;
      O     "PUSHER_RAM_DB".PUSH_DRV_FWD_CMD_PF;
      );
      AN    "PUSHER_RAM_DB".PUSH_RLS_OVN_FACE_RCHD;
      A     "PUSHER_RAM_DB".PUSH_RLS_GUIDE_ENT;
      O;
      A(;
      O     "PUSHER_RAM_DB".PUSH_DRV_REV_CMD;
      O     "PUSHER_RAM_DB".PUSH_DRV_REV_CMD_PF;
      );
      AN    "PUSHER_RAM_DB".PUSH_RLS_OVN_FACE_RCHD;
      );
      =     L 0.2;
      A     L 0.2;
      A     "PUSHER_RAM_DB".PUSH_DRV_PROF_HDWR_SS;
      JNB   _012;
      L     23500;
      T     PQW 262;
_012: NOP   0;
      A     L 0.2;
      AN    "PUSHER_RAM_DB".PUSH_DRV_PROF_HDWR_SS;
      =     L 0.3;
      A     L 0.3;
      A     "PUSHER_RAM_DB".PUSH_DRV_FWD_CMD_PF;
      JNB   _013;
      L     17000;
      T     "PUSHER_RAM_DB".DRV_CONTROL_WORD_2;
_013: NOP   0;
      A     L 0.3;
      A     "PUSHER_RAM_DB".PUSH_DRV_REV_CMD_PF;
      JNB   _014;
      L     -17000;
      T     "PUSHER_RAM_DB".DRV_CONTROL_WORD_2;
_014: NOP   0;
      A     L 0.1;
      A(;
      O     "PUSHER_RAM_DB".PUSH_RLS_OVN_FACE_RCHD;
      O;
      A(;
      O     "PUSHER_RAM_DB".PUSH_DRV_FWD_CMD;
      O     "PUSHER_RAM_DB".PUSH_DRV_FWD_CMD_PF;
      );
      AN    "PUSHER_RAM_DB".PUSH_RLS_GUIDE_ENT;
      );
      =     L 0.2;
      A     L 0.2;
      A     "PUSHER_RAM_DB".PUSH_DRV_PROF_HDWR_SS;
      JNB   _015;
      L     6000;
      T     PQW 262;
_015: NOP   0;
      A     L 0.2;
      AN    "PUSHER_RAM_DB".PUSH_DRV_PROF_HDWR_SS;
      =     L 0.3;
      A     L 0.3;
      A     "PUSHER_RAM_DB".PUSH_DRV_FWD_CMD_PF;
      JNB   _016;
      L     5000;
      T     "PUSHER_RAM_DB".DRV_CONTROL_WORD_2;
_016: NOP   0;
      A     L 0.3;
      A     "PUSHER_RAM_DB".PUSH_DRV_REV_CMD_PF;
      JNB   _017;
      L     -5000;
      T     "PUSHER_RAM_DB".DRV_CONTROL_WORD_2;
_017: NOP   0;
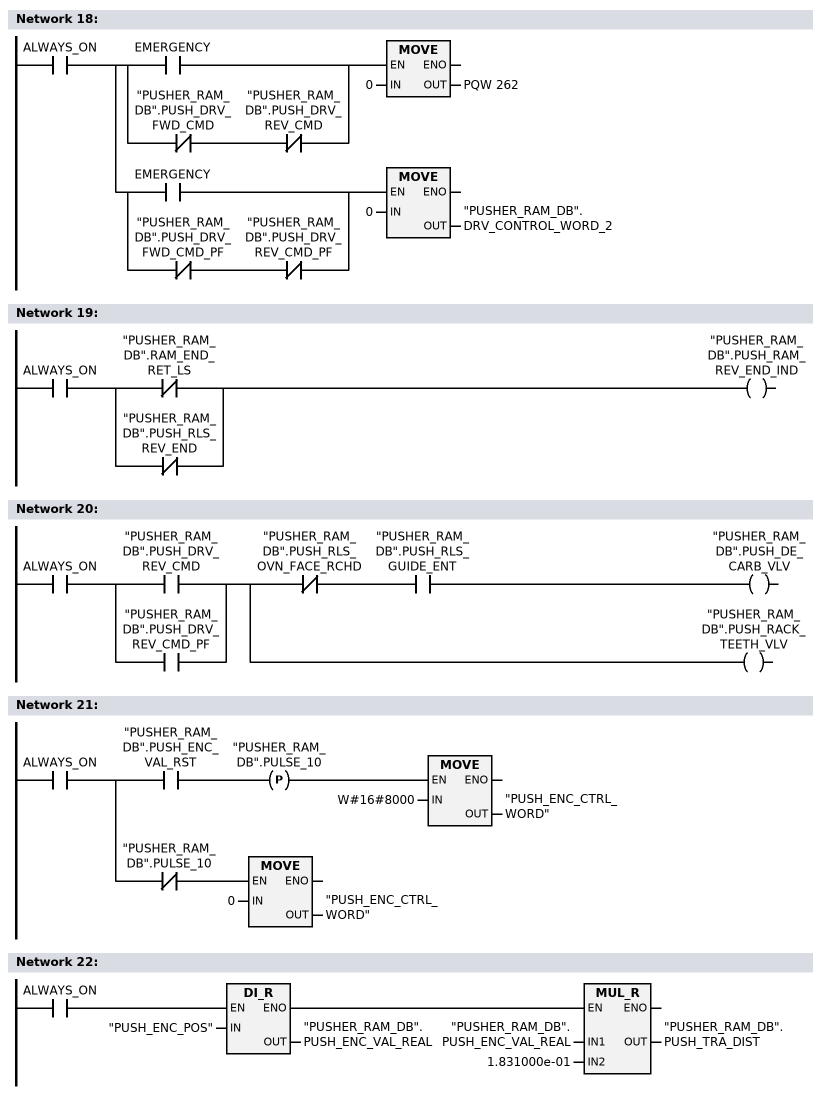
NETWORK
TITLE =
      A     "ALWAYS_ON";
      =     L 0.0;
      A     L 0.0;
      A(;
      O     "EMERGENCY";
      O;
      AN    "PUSHER_RAM_DB".PUSH_DRV_FWD_CMD;
      AN    "PUSHER_RAM_DB".PUSH_DRV_REV_CMD;
      );
      JNB   _018;
      L     0;
      T     PQW 262;
_018: NOP   0;
      A     L 0.0;
      A(;
      O     "EMERGENCY";
      O;
      AN    "PUSHER_RAM_DB".PUSH_DRV_FWD_CMD_PF;
      AN    "PUSHER_RAM_DB".PUSH_DRV_REV_CMD_PF;
      );
      JNB   _019;
      L     0;
      T     "PUSHER_RAM_DB".DRV_CONTROL_WORD_2;
_019: NOP   0;
NETWORK
TITLE =
      A     "ALWAYS_ON";
      A(;
      ON    "PUSHER_RAM_DB".RAM_END_RET_LS;
      ON    "PUSHER_RAM_DB".PUSH_RLS_REV_END;
      );
      =     "PUSHER_RAM_DB".PUSH_RAM_REV_END_IND;
NETWORK
TITLE =
      A     "ALWAYS_ON";
      A(;
      O     "PUSHER_RAM_DB".PUSH_DRV_REV_CMD;
      O     "PUSHER_RAM_DB".PUSH_DRV_REV_CMD_PF;
      );
      =     L 0.0;
      A     L 0.0;
      AN    "PUSHER_RAM_DB".PUSH_RLS_OVN_FACE_RCHD;
      A     "PUSHER_RAM_DB".PUSH_RLS_GUIDE_ENT;
      =     "PUSHER_RAM_DB".PUSH_DE_CARB_VLV;
      A     L 0.0;
      BLD   102;
      =     "PUSHER_RAM_DB".PUSH_RACK_TEETH_VLV;
NETWORK
TITLE =
      A     "ALWAYS_ON";
      =     L 0.0;
      A     L 0.0;
      A     "PUSHER_RAM_DB".PUSH_ENC_VAL_RST;
      FP    "PUSHER_RAM_DB".PULSE_10;
      JNB   _01a;
      L     W#16#8000;
      T     "PUSH_ENC_CTRL_WORD";
_01a: NOP   0;
      A     L 0.0;
      AN    "PUSHER_RAM_DB".PULSE_10;
      JNB   _01b;
      L     0;
      T     "PUSH_ENC_CTRL_WORD";
_01b: NOP   0;
NETWORK
TITLE =
      A(;
      A     "ALWAYS_ON";
      JNB   _01c;
      L     "PUSH_ENC_POS";
      DTR;
      T     "PUSHER_RAM_DB".PUSH_ENC_VAL_REAL;
      SET;
      SAVE;
      CLR;
_01c: A     BR;
      );
      JNB   _01d;
      L     "PUSHER_RAM_DB".PUSH_ENC_VAL_REAL;
      L     1.831000e-01;
      *R;
      T     "PUSHER_RAM_DB".PUSH_TRA_DIST;
_01d: NOP   0;
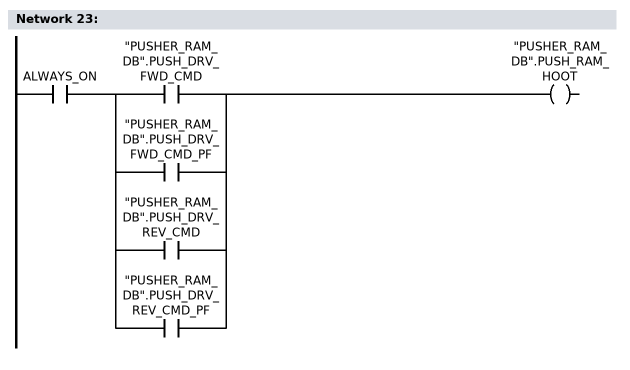
NETWORK
TITLE =
      A     "ALWAYS_ON";
      A(;
      O     "PUSHER_RAM_DB".PUSH_DRV_FWD_CMD;
      O     "PUSHER_RAM_DB".PUSH_DRV_FWD_CMD_PF;
      O     "PUSHER_RAM_DB".PUSH_DRV_REV_CMD;
      O     "PUSHER_RAM_DB".PUSH_DRV_REV_CMD_PF;
      );
      =     "PUSHER_RAM_DB".PUSH_RAM_HOOT;
END_FUNCTION

FUNCTION "AIR_COMPRESSOR" : VOID	// FC 9
AUTHOR : Kamillas
VERSION : 0.1
BEGIN
// (block stored without names or comments; labels and parameter names are numbered)
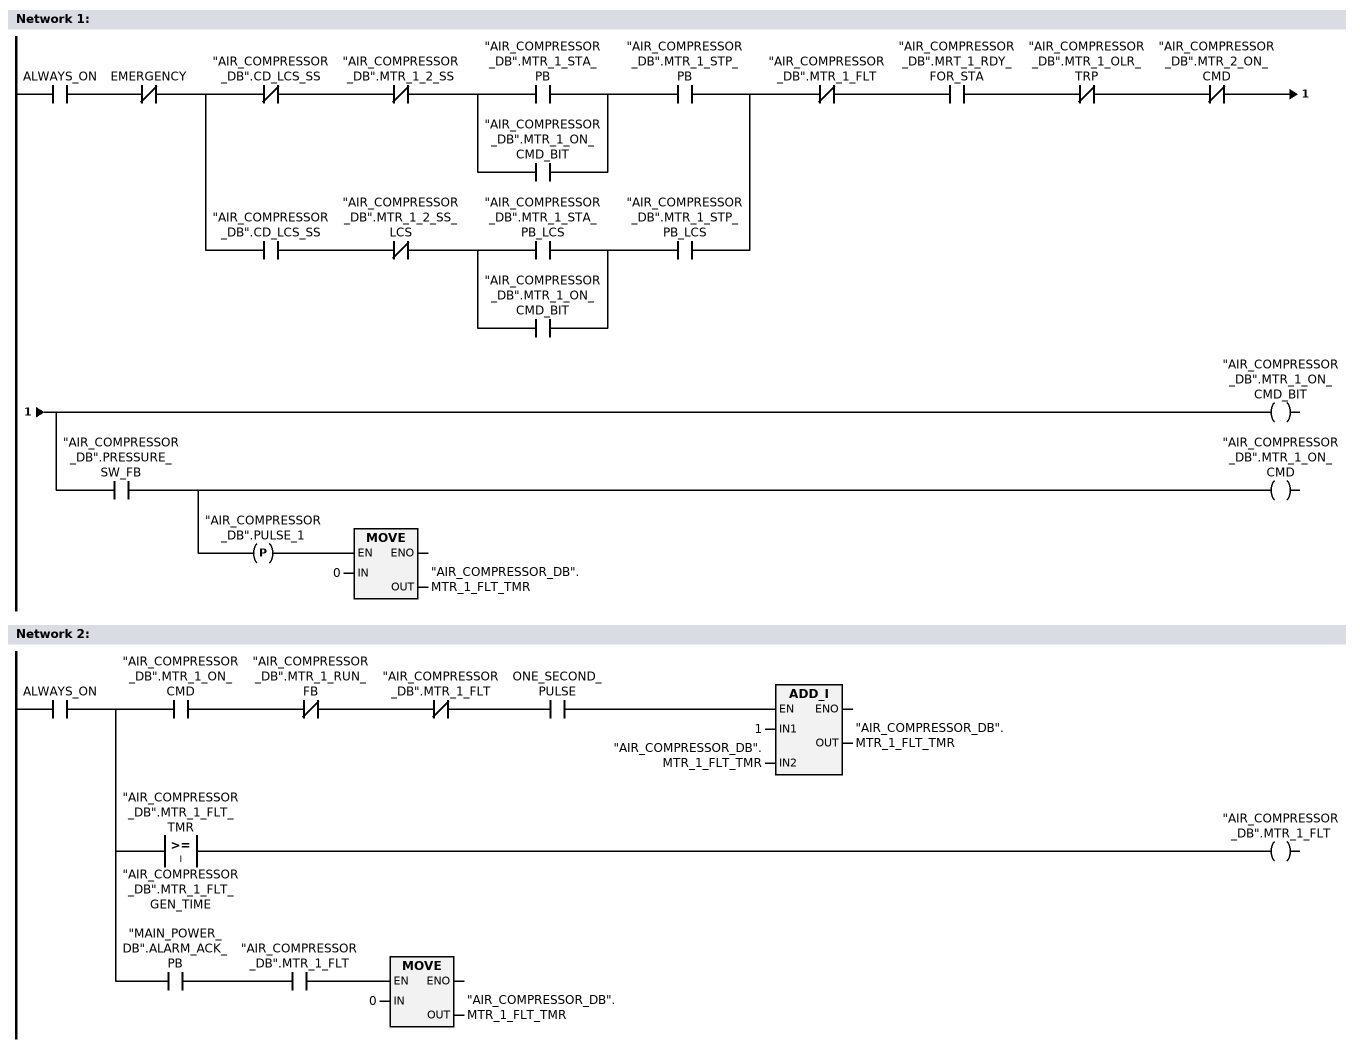
NETWORK
TITLE =
      A     "ALWAYS_ON";
      AN    "EMERGENCY";
      A(;
      AN    "AIR_COMPRESSOR_DB".CD_LCS_SS;
      AN    "AIR_COMPRESSOR_DB".MTR_1_2_SS;
      A(;
      O     "AIR_COMPRESSOR_DB".MTR_1_STA_PB;
      O     "AIR_COMPRESSOR_DB".MTR_1_ON_CMD_BIT;
      );
      A     "AIR_COMPRESSOR_DB".MTR_1_STP_PB;
      O;
      A     "AIR_COMPRESSOR_DB".CD_LCS_SS;
      AN    "AIR_COMPRESSOR_DB".MTR_1_2_SS_LCS;
      A(;
      O     "AIR_COMPRESSOR_DB".MTR_1_STA_PB_LCS;
      O     "AIR_COMPRESSOR_DB".MTR_1_ON_CMD_BIT;
      );
      A     "AIR_COMPRESSOR_DB".MTR_1_STP_PB_LCS;
      );
      AN    "AIR_COMPRESSOR_DB".MTR_1_FLT;
      A     "AIR_COMPRESSOR_DB".MRT_1_RDY_FOR_STA;
      AN    "AIR_COMPRESSOR_DB".MTR_1_OLR_TRP;
      AN    "AIR_COMPRESSOR_DB".MTR_2_ON_CMD;
      =     L 0.0;
      A     L 0.0;
      BLD   102;
      =     "AIR_COMPRESSOR_DB".MTR_1_ON_CMD_BIT;
      A     L 0.0;
      A     "AIR_COMPRESSOR_DB".PRESSURE_SW_FB;
      =     L 0.1;
      A     L 0.1;
      BLD   102;
      =     "AIR_COMPRESSOR_DB".MTR_1_ON_CMD;
      A     L 0.1;
      FP    "AIR_COMPRESSOR_DB".PULSE_1;
      JNB   M001;
      L     0;
      T     "AIR_COMPRESSOR_DB".MTR_1_FLT_TMR;
M001: NOP   0;
NETWORK
TITLE =
      A     "ALWAYS_ON";
      =     L 0.0;
      A     L 0.0;
      A     "AIR_COMPRESSOR_DB".MTR_1_ON_CMD;
      AN    "AIR_COMPRESSOR_DB".MTR_1_RUN_FB;
      AN    "AIR_COMPRESSOR_DB".MTR_1_FLT;
      A     "ONE_SECOND_PULSE";
      JNB   M002;
      L     1;
      L     "AIR_COMPRESSOR_DB".MTR_1_FLT_TMR;
      +I;
      T     "AIR_COMPRESSOR_DB".MTR_1_FLT_TMR;
M002: NOP   0;
      A     L 0.0;
      A(;
      L     "AIR_COMPRESSOR_DB".MTR_1_FLT_TMR;
      L     "AIR_COMPRESSOR_DB".MTR_1_FLT_GEN_TIME;
      >=I;
      );
      =     "AIR_COMPRESSOR_DB".MTR_1_FLT;
      A     L 0.0;
      A     "MAIN_POWER_DB".ALARM_ACK_PB;
      A     "AIR_COMPRESSOR_DB".MTR_1_FLT;
      JNB   M003;
      L     0;
      T     "AIR_COMPRESSOR_DB".MTR_1_FLT_TMR;
M003: NOP   0;
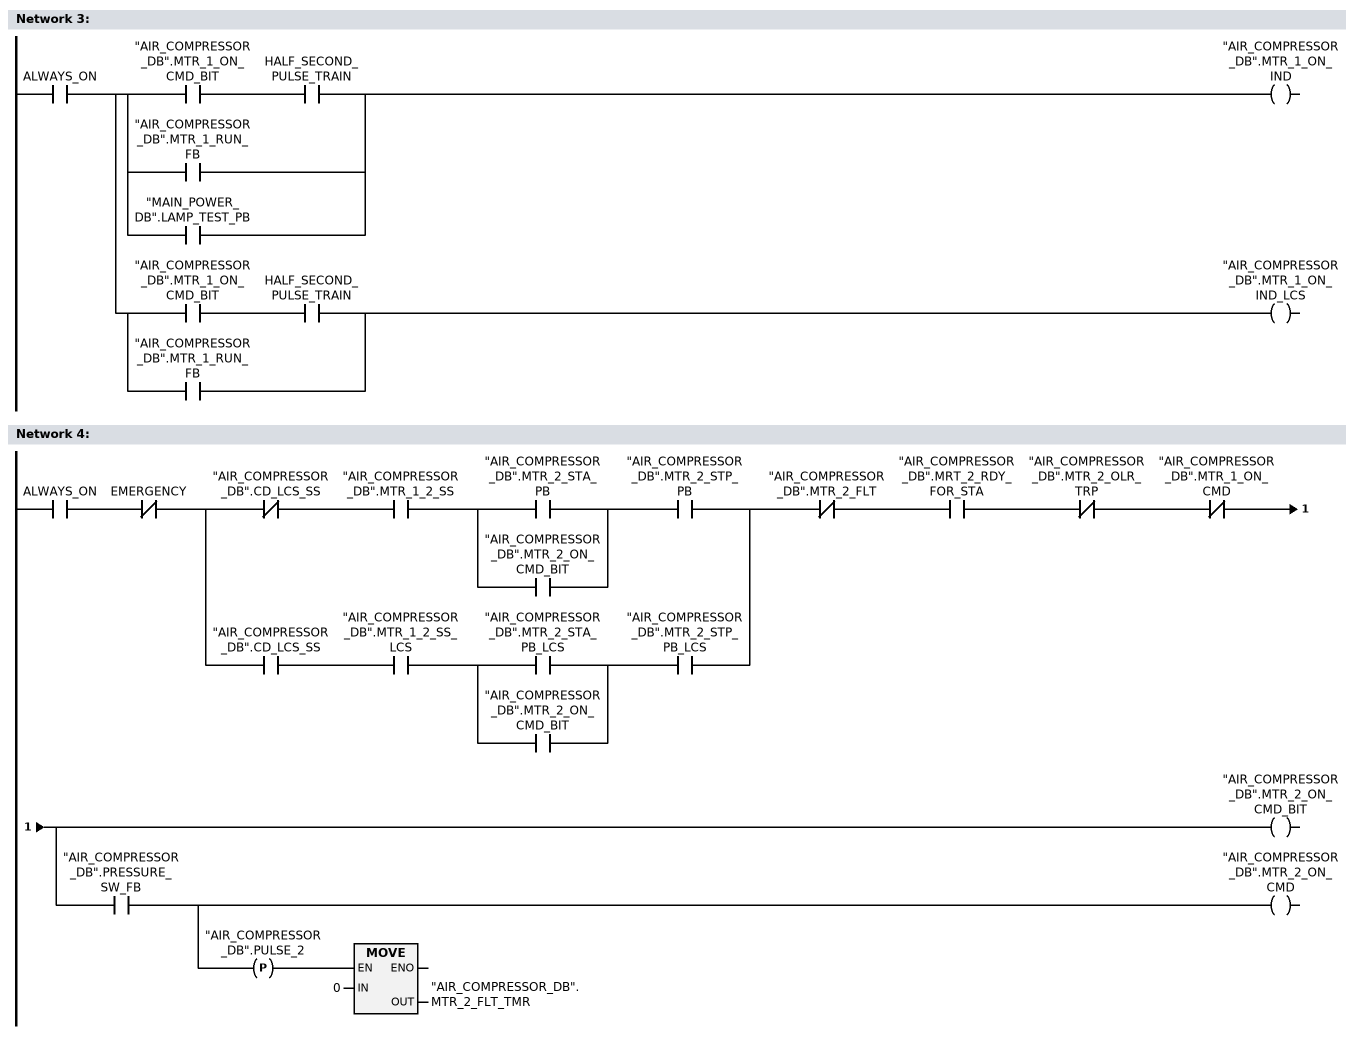
NETWORK
TITLE =
      A     "ALWAYS_ON";
      =     L 0.0;
      A     L 0.0;
      A(;
      A     "AIR_COMPRESSOR_DB".MTR_1_ON_CMD_BIT;
      A     "HALF_SECOND_PULSE_TRAIN";
      O     "AIR_COMPRESSOR_DB".MTR_1_RUN_FB;
      O     "MAIN_POWER_DB".LAMP_TEST_PB;
      );
      =     "AIR_COMPRESSOR_DB".MTR_1_ON_IND;
      A     L 0.0;
      A(;
      A     "AIR_COMPRESSOR_DB".MTR_1_ON_CMD_BIT;
      A     "HALF_SECOND_PULSE_TRAIN";
      O     "AIR_COMPRESSOR_DB".MTR_1_RUN_FB;
      );
      =     "AIR_COMPRESSOR_DB".MTR_1_ON_IND_LCS;
NETWORK
TITLE =
      A     "ALWAYS_ON";
      AN    "EMERGENCY";
      A(;
      AN    "AIR_COMPRESSOR_DB".CD_LCS_SS;
      A     "AIR_COMPRESSOR_DB".MTR_1_2_SS;
      A(;
      O     "AIR_COMPRESSOR_DB".MTR_2_STA_PB;
      O     "AIR_COMPRESSOR_DB".MTR_2_ON_CMD_BIT;
      );
      A     "AIR_COMPRESSOR_DB".MTR_2_STP_PB;
      O;
      A     "AIR_COMPRESSOR_DB".CD_LCS_SS;
      A     "AIR_COMPRESSOR_DB".MTR_1_2_SS_LCS;
      A(;
      O     "AIR_COMPRESSOR_DB".MTR_2_STA_PB_LCS;
      O     "AIR_COMPRESSOR_DB".MTR_2_ON_CMD_BIT;
      );
      A     "AIR_COMPRESSOR_DB".MTR_2_STP_PB_LCS;
      );
      AN    "AIR_COMPRESSOR_DB".MTR_2_FLT;
      A     "AIR_COMPRESSOR_DB".MRT_2_RDY_FOR_STA;
      AN    "AIR_COMPRESSOR_DB".MTR_2_OLR_TRP;
      AN    "AIR_COMPRESSOR_DB".MTR_1_ON_CMD;
      =     L 0.0;
      A     L 0.0;
      BLD   102;
      =     "AIR_COMPRESSOR_DB".MTR_2_ON_CMD_BIT;
      A     L 0.0;
      A     "AIR_COMPRESSOR_DB".PRESSURE_SW_FB;
      =     L 0.1;
      A     L 0.1;
      BLD   102;
      =     "AIR_COMPRESSOR_DB".MTR_2_ON_CMD;
      A     L 0.1;
      FP    "AIR_COMPRESSOR_DB".PULSE_2;
      JNB   M004;
      L     0;
      T     "AIR_COMPRESSOR_DB".MTR_2_FLT_TMR;
M004: NOP   0;
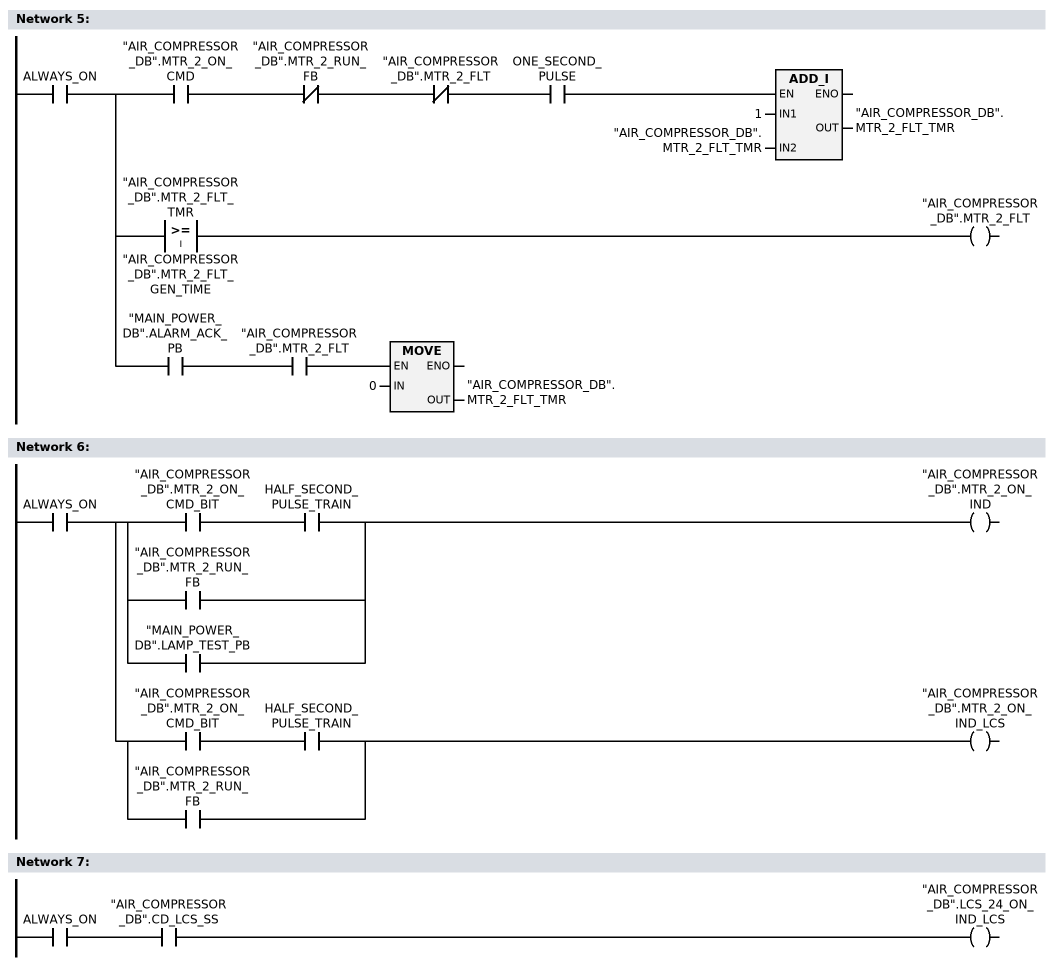
NETWORK
TITLE =
      A     "ALWAYS_ON";
      =     L 0.0;
      A     L 0.0;
      A     "AIR_COMPRESSOR_DB".MTR_2_ON_CMD;
      AN    "AIR_COMPRESSOR_DB".MTR_2_RUN_FB;
      AN    "AIR_COMPRESSOR_DB".MTR_2_FLT;
      A     "ONE_SECOND_PULSE";
      JNB   M005;
      L     1;
      L     "AIR_COMPRESSOR_DB".MTR_2_FLT_TMR;
      +I;
      T     "AIR_COMPRESSOR_DB".MTR_2_FLT_TMR;
M005: NOP   0;
      A     L 0.0;
      A(;
      L     "AIR_COMPRESSOR_DB".MTR_2_FLT_TMR;
      L     "AIR_COMPRESSOR_DB".MTR_2_FLT_GEN_TIME;
      >=I;
      );
      =     "AIR_COMPRESSOR_DB".MTR_2_FLT;
      A     L 0.0;
      A     "MAIN_POWER_DB".ALARM_ACK_PB;
      A     "AIR_COMPRESSOR_DB".MTR_2_FLT;
      JNB   M006;
      L     0;
      T     "AIR_COMPRESSOR_DB".MTR_2_FLT_TMR;
M006: NOP   0;
NETWORK
TITLE =
      A     "ALWAYS_ON";
      =     L 0.0;
      A     L 0.0;
      A(;
      A     "AIR_COMPRESSOR_DB".MTR_2_ON_CMD_BIT;
      A     "HALF_SECOND_PULSE_TRAIN";
      O     "AIR_COMPRESSOR_DB".MTR_2_RUN_FB;
      O     "MAIN_POWER_DB".LAMP_TEST_PB;
      );
      =     "AIR_COMPRESSOR_DB".MTR_2_ON_IND;
      A     L 0.0;
      A(;
      A     "AIR_COMPRESSOR_DB".MTR_2_ON_CMD_BIT;
      A     "HALF_SECOND_PULSE_TRAIN";
      O     "AIR_COMPRESSOR_DB".MTR_2_RUN_FB;
      );
      =     "AIR_COMPRESSOR_DB".MTR_2_ON_IND_LCS;
NETWORK
TITLE =
      A     "ALWAYS_ON";
      A     "AIR_COMPRESSOR_DB".CD_LCS_SS;
      =     "AIR_COMPRESSOR_DB".LCS_24_ON_IND_LCS;
END_FUNCTION

FUNCTION "DOOR_AND_JAMB" : VOID	// FC 10
AUTHOR : Kamillas
VERSION : 0.1
BEGIN
// (block stored without names or comments; labels and parameter names are numbered)
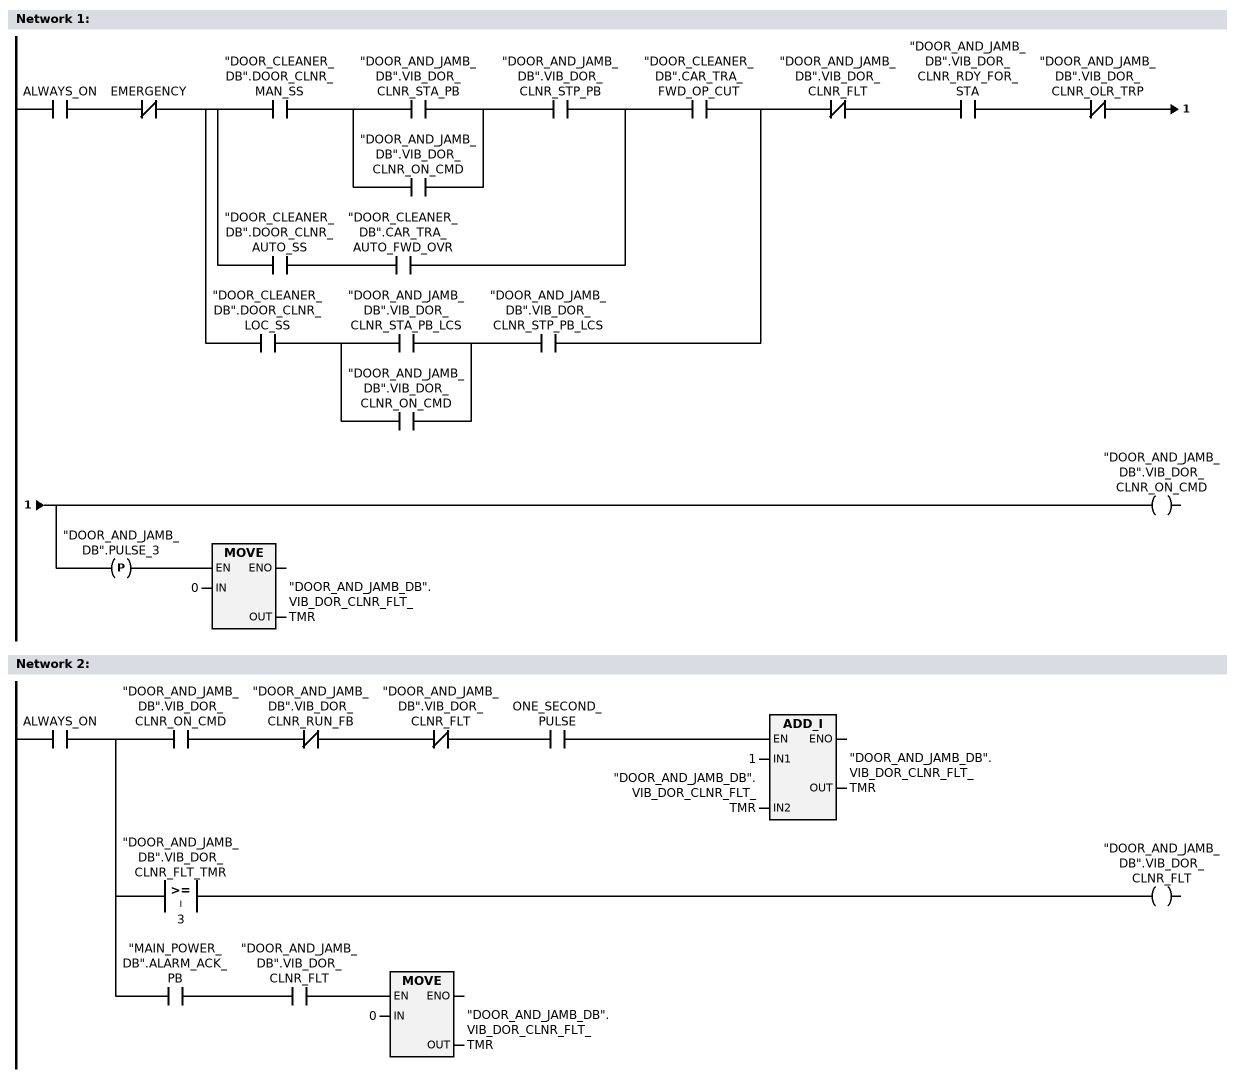
NETWORK
TITLE =
      A     "ALWAYS_ON";
      AN    "EMERGENCY";
      A(;
      A(;
      A     "DOOR_CLEANER_DB".DOOR_CLNR_MAN_SS;
      A(;
      O     "DOOR_AND_JAMB_DB".VIB_DOR_CLNR_STA_PB;
      O     "DOOR_AND_JAMB_DB".VIB_DOR_CLNR_ON_CMD;
      );
      A     "DOOR_AND_JAMB_DB".VIB_DOR_CLNR_STP_PB;
      O;
      A     "DOOR_CLEANER_DB".DOOR_CLNR_AUTO_SS;
      A     "DOOR_CLEANER_DB".CAR_TRA_AUTO_FWD_OVR;
      );
      A     "DOOR_CLEANER_DB".CAR_TRA_FWD_OP_CUT;
      O;
      A     "DOOR_CLEANER_DB".DOOR_CLNR_LOC_SS;
      A(;
      O     "DOOR_AND_JAMB_DB".VIB_DOR_CLNR_STA_PB_LCS;
      O     "DOOR_AND_JAMB_DB".VIB_DOR_CLNR_ON_CMD;
      );
      A     "DOOR_AND_JAMB_DB".VIB_DOR_CLNR_STP_PB_LCS;
      );
      AN    "DOOR_AND_JAMB_DB".VIB_DOR_CLNR_FLT;
      A     "DOOR_AND_JAMB_DB".VIB_DOR_CLNR_RDY_FOR_STA;
      AN    "DOOR_AND_JAMB_DB".VIB_DOR_CLNR_OLR_TRP;
      =     L 0.0;
      A     L 0.0;
      BLD   102;
      =     "DOOR_AND_JAMB_DB".VIB_DOR_CLNR_ON_CMD;
      A     L 0.0;
      FP    "DOOR_AND_JAMB_DB".PULSE_3;
      JNB   M001;
      L     0;
      T     "DOOR_AND_JAMB_DB".VIB_DOR_CLNR_FLT_TMR;
M001: NOP   0;
NETWORK
TITLE =
      A     "ALWAYS_ON";
      =     L 0.0;
      A     L 0.0;
      A     "DOOR_AND_JAMB_DB".VIB_DOR_CLNR_ON_CMD;
      AN    "DOOR_AND_JAMB_DB".VIB_DOR_CLNR_RUN_FB;
      AN    "DOOR_AND_JAMB_DB".VIB_DOR_CLNR_FLT;
      A     "ONE_SECOND_PULSE";
      JNB   M002;
      L     1;
      L     "DOOR_AND_JAMB_DB".VIB_DOR_CLNR_FLT_TMR;
      +I;
      T     "DOOR_AND_JAMB_DB".VIB_DOR_CLNR_FLT_TMR;
M002: NOP   0;
      A     L 0.0;
      A(;
      L     "DOOR_AND_JAMB_DB".VIB_DOR_CLNR_FLT_TMR;
      L     3;
      >=I;
      );
      =     "DOOR_AND_JAMB_DB".VIB_DOR_CLNR_FLT;
      A     L 0.0;
      A     "MAIN_POWER_DB".ALARM_ACK_PB;
      A     "DOOR_AND_JAMB_DB".VIB_DOR_CLNR_FLT;
      JNB   M003;
      L     0;
      T     "DOOR_AND_JAMB_DB".VIB_DOR_CLNR_FLT_TMR;
M003: NOP   0;
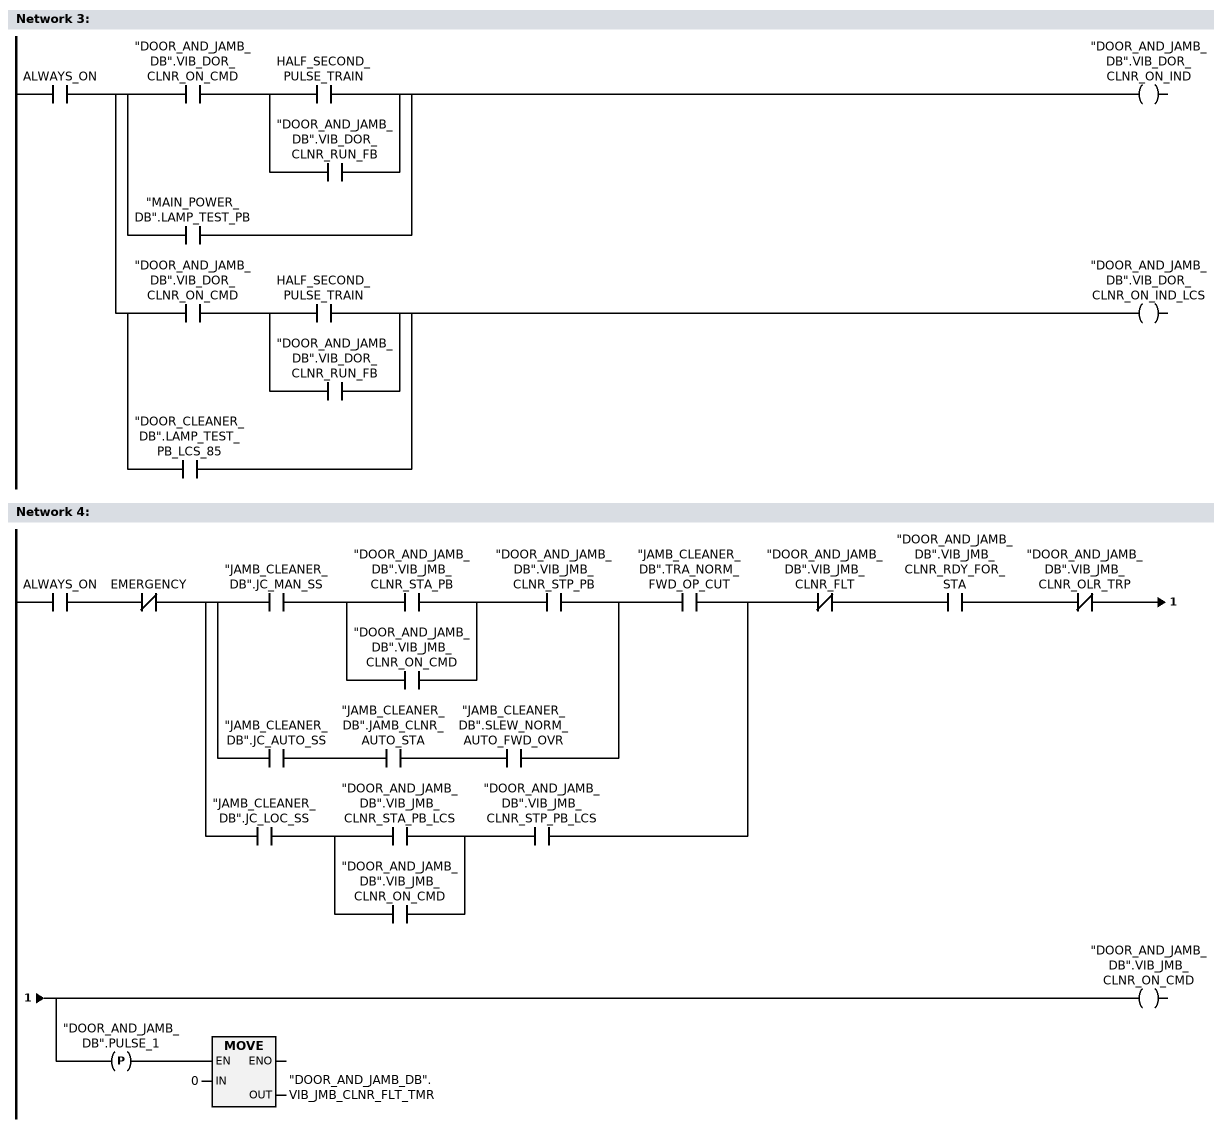
NETWORK
TITLE =
      A     "ALWAYS_ON";
      =     L 0.0;
      A     L 0.0;
      A(;
      A     "DOOR_AND_JAMB_DB".VIB_DOR_CLNR_ON_CMD;
      A(;
      O     "HALF_SECOND_PULSE_TRAIN";
      O     "DOOR_AND_JAMB_DB".VIB_DOR_CLNR_RUN_FB;
      );
      O     "MAIN_POWER_DB".LAMP_TEST_PB;
      );
      =     "DOOR_AND_JAMB_DB".VIB_DOR_CLNR_ON_IND;
      A     L 0.0;
      A(;
      A     "DOOR_AND_JAMB_DB".VIB_DOR_CLNR_ON_CMD;
      A(;
      O     "HALF_SECOND_PULSE_TRAIN";
      O     "DOOR_AND_JAMB_DB".VIB_DOR_CLNR_RUN_FB;
      );
      O     "DOOR_CLEANER_DB".LAMP_TEST_PB_LCS_85;
      );
      =     "DOOR_AND_JAMB_DB".VIB_DOR_CLNR_ON_IND_LCS;
NETWORK
TITLE =
      A     "ALWAYS_ON";
      AN    "EMERGENCY";
      A(;
      A(;
      A     "JAMB_CLEANER_DB".JC_MAN_SS;
      A(;
      O     "DOOR_AND_JAMB_DB".VIB_JMB_CLNR_STA_PB;
      O     "DOOR_AND_JAMB_DB".VIB_JMB_CLNR_ON_CMD;
      );
      A     "DOOR_AND_JAMB_DB".VIB_JMB_CLNR_STP_PB;
      O;
      A     "JAMB_CLEANER_DB".JC_AUTO_SS;
      A     "JAMB_CLEANER_DB".JAMB_CLNR_AUTO_STA;
      A     "JAMB_CLEANER_DB".SLEW_NORM_AUTO_FWD_OVR;
      );
      A     "JAMB_CLEANER_DB".TRA_NORM_FWD_OP_CUT;
      O;
      A     "JAMB_CLEANER_DB".JC_LOC_SS;
      A(;
      O     "DOOR_AND_JAMB_DB".VIB_JMB_CLNR_STA_PB_LCS;
      O     "DOOR_AND_JAMB_DB".VIB_JMB_CLNR_ON_CMD;
      );
      A     "DOOR_AND_JAMB_DB".VIB_JMB_CLNR_STP_PB_LCS;
      );
      AN    "DOOR_AND_JAMB_DB".VIB_JMB_CLNR_FLT;
      A     "DOOR_AND_JAMB_DB".VIB_JMB_CLNR_RDY_FOR_STA;
      AN    "DOOR_AND_JAMB_DB".VIB_JMB_CLNR_OLR_TRP;
      =     L 0.0;
      A     L 0.0;
      BLD   102;
      =     "DOOR_AND_JAMB_DB".VIB_JMB_CLNR_ON_CMD;
      A     L 0.0;
      FP    "DOOR_AND_JAMB_DB".PULSE_1;
      JNB   M004;
      L     0;
      T     "DOOR_AND_JAMB_DB".VIB_JMB_CLNR_FLT_TMR;
M004: NOP   0;
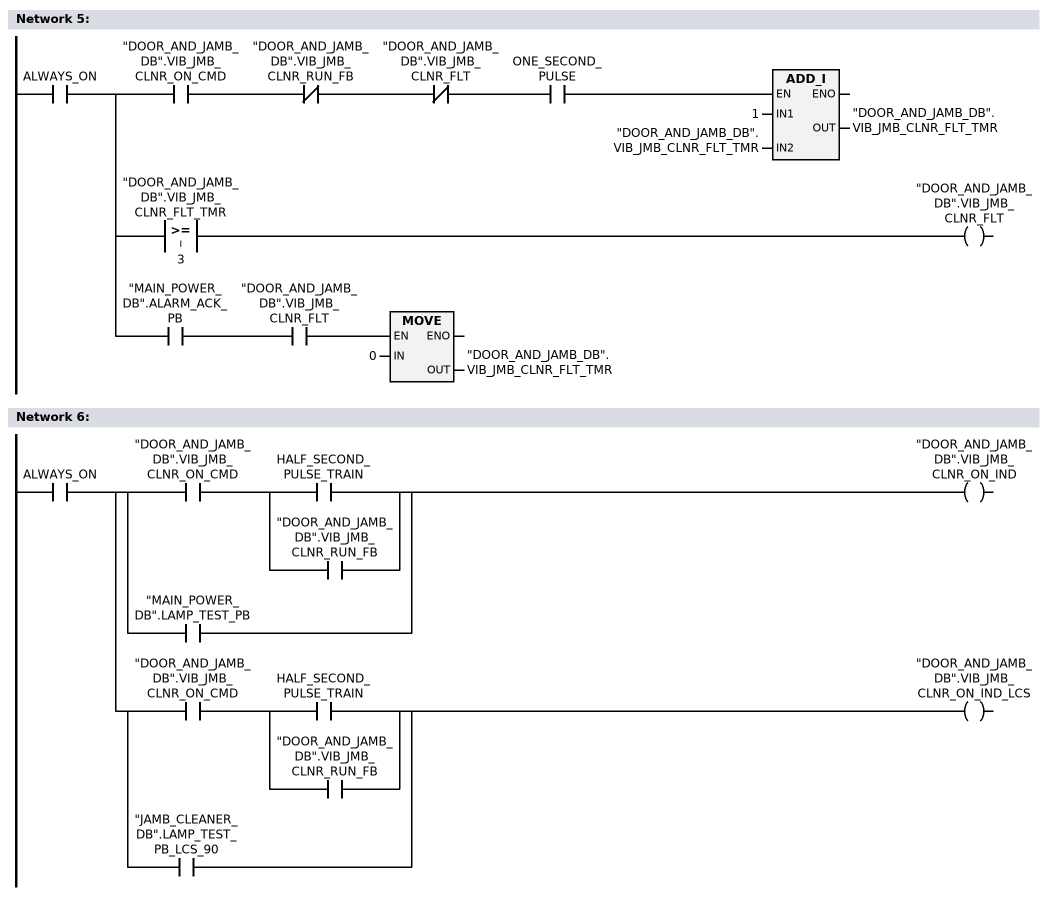
NETWORK
TITLE =
      A     "ALWAYS_ON";
      =     L 0.0;
      A     L 0.0;
      A     "DOOR_AND_JAMB_DB".VIB_JMB_CLNR_ON_CMD;
      AN    "DOOR_AND_JAMB_DB".VIB_JMB_CLNR_RUN_FB;
      AN    "DOOR_AND_JAMB_DB".VIB_JMB_CLNR_FLT;
      A     "ONE_SECOND_PULSE";
      JNB   M005;
      L     1;
      L     "DOOR_AND_JAMB_DB".VIB_JMB_CLNR_FLT_TMR;
      +I;
      T     "DOOR_AND_JAMB_DB".VIB_JMB_CLNR_FLT_TMR;
M005: NOP   0;
      A     L 0.0;
      A(;
      L     "DOOR_AND_JAMB_DB".VIB_JMB_CLNR_FLT_TMR;
      L     3;
      >=I;
      );
      =     "DOOR_AND_JAMB_DB".VIB_JMB_CLNR_FLT;
      A     L 0.0;
      A     "MAIN_POWER_DB".ALARM_ACK_PB;
      A     "DOOR_AND_JAMB_DB".VIB_JMB_CLNR_FLT;
      JNB   M006;
      L     0;
      T     "DOOR_AND_JAMB_DB".VIB_JMB_CLNR_FLT_TMR;
M006: NOP   0;
NETWORK
TITLE =
      A     "ALWAYS_ON";
      =     L 0.0;
      A     L 0.0;
      A(;
      A     "DOOR_AND_JAMB_DB".VIB_JMB_CLNR_ON_CMD;
      A(;
      O     "HALF_SECOND_PULSE_TRAIN";
      O     "DOOR_AND_JAMB_DB".VIB_JMB_CLNR_RUN_FB;
      );
      O     "MAIN_POWER_DB".LAMP_TEST_PB;
      );
      =     "DOOR_AND_JAMB_DB".VIB_JMB_CLNR_ON_IND;
      A     L 0.0;
      A(;
      A     "DOOR_AND_JAMB_DB".VIB_JMB_CLNR_ON_CMD;
      A(;
      O     "HALF_SECOND_PULSE_TRAIN";
      O     "DOOR_AND_JAMB_DB".VIB_JMB_CLNR_RUN_FB;
      );
      O     "JAMB_CLEANER_DB".LAMP_TEST_PB_LCS_90;
      );
      =     "DOOR_AND_JAMB_DB".VIB_JMB_CLNR_ON_IND_LCS;
END_FUNCTION

FUNCTION "LEVELER_BLOWER" : VOID	// FC 11
AUTHOR : Kamillas
VERSION : 0.1
BEGIN
// (block stored without names or comments; labels and parameter names are numbered)
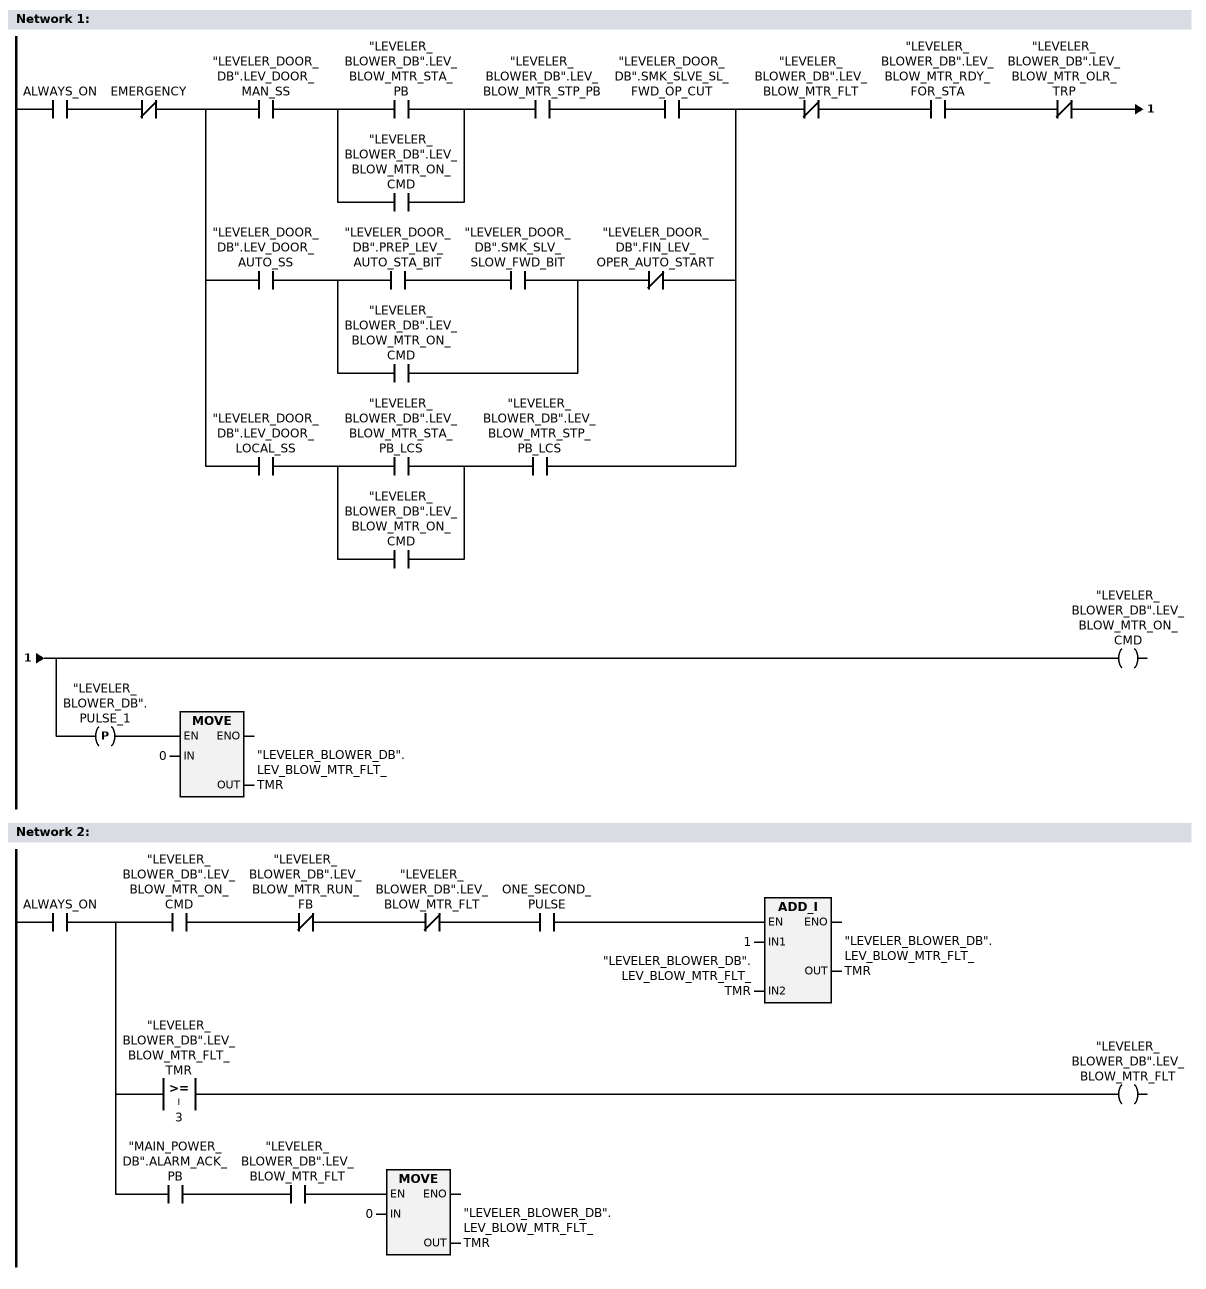
NETWORK
TITLE =
      A     "ALWAYS_ON";
      AN    "EMERGENCY";
      A(;
      A     "LEVELER_DOOR_DB".LEV_DOOR_MAN_SS;
      A(;
      O     "LEVELER_BLOWER_DB".LEV_BLOW_MTR_STA_PB;
      O     "LEVELER_BLOWER_DB".LEV_BLOW_MTR_ON_CMD;
      );
      A     "LEVELER_BLOWER_DB".LEV_BLOW_MTR_STP_PB;
      A     "LEVELER_DOOR_DB".SMK_SLVE_SL_FWD_OP_CUT;
      O;
      A     "LEVELER_DOOR_DB".LEV_DOOR_AUTO_SS;
      A(;
      A     "LEVELER_DOOR_DB".PREP_LEV_AUTO_STA_BIT;
      A     "LEVELER_DOOR_DB".SMK_SLV_SLOW_FWD_BIT;
      O     "LEVELER_BLOWER_DB".LEV_BLOW_MTR_ON_CMD;
      );
      AN    "LEVELER_DOOR_DB".FIN_LEV_OPER_AUTO_START;
      O;
      A     "LEVELER_DOOR_DB".LEV_DOOR_LOCAL_SS;
      A(;
      O     "LEVELER_BLOWER_DB".LEV_BLOW_MTR_STA_PB_LCS;
      O     "LEVELER_BLOWER_DB".LEV_BLOW_MTR_ON_CMD;
      );
      A     "LEVELER_BLOWER_DB".LEV_BLOW_MTR_STP_PB_LCS;
      );
      AN    "LEVELER_BLOWER_DB".LEV_BLOW_MTR_FLT;
      A     "LEVELER_BLOWER_DB".LEV_BLOW_MTR_RDY_FOR_STA;
      AN    "LEVELER_BLOWER_DB".LEV_BLOW_MTR_OLR_TRP;
      =     L 0.0;
      A     L 0.0;
      BLD   102;
      =     "LEVELER_BLOWER_DB".LEV_BLOW_MTR_ON_CMD;
      A     L 0.0;
      FP    "LEVELER_BLOWER_DB".PULSE_1;
      JNB   M001;
      L     0;
      T     "LEVELER_BLOWER_DB".LEV_BLOW_MTR_FLT_TMR;
M001: NOP   0;
NETWORK
TITLE =
      A     "ALWAYS_ON";
      =     L 0.0;
      A     L 0.0;
      A     "LEVELER_BLOWER_DB".LEV_BLOW_MTR_ON_CMD;
      AN    "LEVELER_BLOWER_DB".LEV_BLOW_MTR_RUN_FB;
      AN    "LEVELER_BLOWER_DB".LEV_BLOW_MTR_FLT;
      A     "ONE_SECOND_PULSE";
      JNB   M002;
      L     1;
      L     "LEVELER_BLOWER_DB".LEV_BLOW_MTR_FLT_TMR;
      +I;
      T     "LEVELER_BLOWER_DB".LEV_BLOW_MTR_FLT_TMR;
M002: NOP   0;
      A     L 0.0;
      A(;
      L     "LEVELER_BLOWER_DB".LEV_BLOW_MTR_FLT_TMR;
      L     3;
      >=I;
      );
      =     "LEVELER_BLOWER_DB".LEV_BLOW_MTR_FLT;
      A     L 0.0;
      A     "MAIN_POWER_DB".ALARM_ACK_PB;
      A     "LEVELER_BLOWER_DB".LEV_BLOW_MTR_FLT;
      JNB   M003;
      L     0;
      T     "LEVELER_BLOWER_DB".LEV_BLOW_MTR_FLT_TMR;
M003: NOP   0;
